# B&R Automation Studio project Soiled_PLC (part 10)

#### Param_1_5kwStar.dat
```
(********************************************************************
 * COPYRIGHT --
 ********************************************************************
 * Data object: Param_1_5kwStar
 * File: Param_1_5kwStar.dat
 * Author:  D.Jefferys
 * Created: October 2, 2009
 ********************************************************************
 * Data object file: Param_1_5kwStar.dat
 ********************************************************************)

;Version 2.00 18/10/2010 D.J. Added 14-26 Trip Delay - Disabled, Changed 14-10 from 3 (Coasting) to 5 (Kenetic Backup + Trip)
;Version 3.00 03/11/2010 D.J. Added CAN Switch Settings
;Version 4.00 02/11/2011 D.J. Added Parameter 40 - Hand on Key on LCP now Disabled

;CAN Module Switch Settings
;--------------------------

;Baudrate
;8 on  7 on  Par 10-01
;8 on  7 off 500kbps
;8 off 7 on  250kbps
;8 off 7 off 125kbps

;Node Number Binary
;1 = 1s
;2 = 2s
;3 = 4s
;4 = 8s
;5 = 16s
;6 = 32s

;
;	!!! DO NOT CHANGE THE SEQUENCE OF THE PARAMETERS
;
; FU parameter to the Ubertragung (only parameter, which deviates from the default values)
;
; 1.5 kW Star
;
; Index, Subindex, Datatype (Bytes), Setting (DINT) ; Comments
0002,00,01,00000001	; [000] 00-02, Motor Speed 0 - RPM, 1 - Hz
0001,00,01,00000000	; [001] 00-01, Language 0 - English, 1 - German
0011,00,01,00000001	; [002] 00-11, Edit Setup 1
0190,00,01,00000000	; [003] 01-90, Motor Thermal Protection, 2 - Thermistor
0040,00,01,00000000 ; [---] 00-40, Hand On Key on LCP 0 - Disabled No Function
0381,00,04,00000050 ; [000] 03-81, QuickStop ramp time 100 - 1s
0458,00,01,00000001	; [004] 04-58, Missing motor phase function, 1 - Trip 100ms
0854,00,01,00000001	; [005] 08-54, Reversing select 1 - Bus only 3 - Bus and Terminal
0211,00,02,00000310	; [006] 02-11, Brake resistor 120 Ohm
0212,00,04,00001200	; [007] 02-12, Brake power limit 1200 Watt
0213,00,01,00000002	; [008] 02-13, Brake check 2 - Alarm
1426,00,01,00000000 ; [---] 14-26, Trip delay at inverter fault 0 = Disabled
0803,00,04,00000002 ; [000] 08-03, Control Word Timeout Time 10 = 1Sec
0804,00,01,00000002	; [009] 08-04, Control Word Timeout Function 2 - Stop with auto restart
0801,00,01,00000002	; [010] 08-01, Control Site, 2 - Controlword only
0223,00,01,00000005	; [011] 02-23, Active brake delay 0,3 s
1761,00,01,00000002	; [012] 17-61, Encoder Signal Monitoring (Encoder faulty), 2 - Trip Changed for testing.
1710,00,01,00000001	; [013] 17-10, Encoder Signal Type 1 - TTL
1711,00,02,00001024	; [014] 17-11, Encoder Resolution 1024 Pulse
0430,00,01,00000001 ; [015] 04-30, Motor Feedback Loss Function, 1 - Warning, 2* - Trip
0431,00,02,00000300 ; [016] 04-31, Motor Feedback Speed Error RPM, 0-600, 300*
0226,00,02,00005000	; [015] 02-26, Torque Ref, 50,00%
0228,00,02,00000200	; [016] 02-28, Gain Boost Factor, 2,00% 0-4% ***************************
0519,00,01,00000003	; [017] 05-19, Terminal 37 Safe Stop, 3 - Safe Stop Warning
0120,00,04,00000150	; [018] 01-20, Motor Power 1.5kW
0101,00,01,00000003	; [019] 01-01, Motor Control Principle, 3 - Flux with motor feedback
0122,00,02,00000400	; [020] 01-22, Motor voltage 400 V
0123,00,02,00000050	; [021] 01-23, Motor frequency 50 Hz
0162,00,02,00000100	; [022] 01-62, Slip compenstation 100%
0410,00,01,00000002	; [023] 04-10, Motor speed direction, 2 - both directions
0540,00,01,00000032	; [024] 05-40, [0] Relay 1 Function, 32 - Mech brake ctrl
0540,01,01,00000032	; [025] 05-40, [1] Relay 2 Function, 32 - Mech brake ctrl
0802,00,01,00000003 ; [---] 08-02, Control Site 3 - Option A CAN Bus
0102,00,01,00000002	; [026] 01-02, Flux Motor Feeback Source 2 - MCB102
0125,00,02,00001400	; [027] 01-25, Motor nominal speed 1440 rpm
0702,00,02,00000070	; [028] 07-02, Speed PID proportionl gain 0,070
0700,00,01,00000002	; [029] 07-00, Speed PID Feedback Source 2 - MCB102
0172,00,01,00000006	; [030] 01-72, Start function, 6 - Hoist Mech. Brake Rel
0210,00,01,00000001	; [031] 02-10, Brake Function, 1 - Resistor brake
1410,00,01,00000005	; [032] 14-10, Mains failure, 3 - Coasting 5 - Kenetic backup , trip
0193,00,01,00000002	; [040] 01-93, Thermistor source, 2 Analogue input 54 Source terminal 50 for 10V //6 - Digital Input 33
0100,00,01,00000001	; [034] 01-00, Configuration mode, 1 - Closed loop with encoder
0139,00,01,00000004	; [035] 01-39, Motor poles, 4
0511,00,01,00000000	; [036] 05-11, Terminal 19, 0 - No Operation
0512,00,01,00000000	; [037] 05-12, Terminal 27, 0 - No Operation
0513,00,01,00000000	; [038] 05-13, Terminal 29, 0 - No Operation
0510,00,01,00000000	; [039] 05-10, Terminal 18, 0 - No Operation
0175,00,02,00000015	; [040] 01-75, Start Speed, 1,5 Hz
0222,00,02,00000005	; [041] 02-22, Activate Brake Speed ?en bei 0,5 Hz
0124,00,04,00000360	; [042] 01-24, Motor current 5,2 A
0341,00,04,00000100	; [043] 03-41, Ramp 1 ramp up time (1 Sec to 50 Hz)
0342,00,04,00000100	; [044] 03-42, Ramp 1 ramp down time (1 Sec to  0 Hz)
0414,00,02,00001000	; [045] 04-14, Motor Speed High Limit 100,0 Hz
0220,00,04,00000180	; [046] 02-20, Release brake current 1,8 A - About Half of motor A?
;0130,00,04,00029763	; [047] 01-30, Stator resistance (Rs) 2,9763 Ohm
;0131,00,04,00022212	; [048] 01-31, Rotor resistance (Rr) 2,2212 Ohm
;0134,00,04,00031036	; [049] 01-34, Rotor leakage reactance (X2) 3,1036 Ohm
;0136,00,04,01803904	; [050] 01-36, Iron loss resistance (Rfe) 1803,904 Ohm
;0135,00,04,00653996	; [051] 01-35, Main reactance (Xh) 65,3996 Ohm
0416,00,02,00002500	; [052] 04-16, Torque limit motor mode, 160,0 - % NOW 250%
0417,00,02,00001600	; [053] 04-17, Torque limit generator mode, 160,0 %
;0133,00,04,00031036	; [054] 01-33, Stator leakage reactance (X1), 3,1036 Ohm
0303,00,04,00100000	; [055] 03-03, Maximum Reference, 100,000
0418,00,04,00001720	; [056] 04-18, Current Limit 172,0 % - NOW 250%
```

### Data object Logical/Robo_Drive_Control/Paramaters_AnaloguePTC/Param_0_25kwStar1 (Simple, version 4.00.0) - Parameters 0.25kW Star Analogue PTC

#### Param_0_25kwStar.dat
```
(********************************************************************
 * COPYRIGHT --
 ********************************************************************
 * Data object: Param_2kwStar
 * File: Param_2kwStar.dat
 * Author:  D.Jefferys
 * Created: February 12, 2009
 ********************************************************************
 * Data object file: Param_2kwStar.dat
 ********************************************************************)

;Version 2.00 18/10/2010 D.J. Added 14-26 Trip Delay - Disabled, Changed 14-10 from 3 (Coasting) to 5 (Kenetic Backup + Trip)
;Version 3.00 03/11/2010 D.J. Added CAN Switch Settings
;Version 4.00 02/11/2011 D.J. Added Parameter 40 - Hand on Key on LCP now Disabled

;CAN Module Switch Settings
;--------------------------

;Baudrate
;8 on  7 on  Par 10-01
;8 on  7 off 500kbps
;8 off 7 on  250kbps
;8 off 7 off 125kbps

;Node Number Binary
;1 = 1s
;2 = 2s
;3 = 4s
;4 = 8s
;5 = 16s
;6 = 32s

;
;	!!! DO NOT CHANGE THE SEQUENCE OF THE PARAMETERS
;
; FU parameter to the Ubertragung (only parameter, which deviates from the default values)
;
; 0.25 kW Star
;
; Index, Subindex, Datatype (Bytes), Setting (DINT) ; Comments
0002,00,01,00000001	; [000] 00-02, Motor Speed 0 - RPM, 1 - Hz
0001,00,01,00000000	; [001] 00-01, Language 0 - English, 1 - German
0011,00,01,00000001	; [002] 00-11, Edit Setup 1
;0190,00,01,00000000	; [003] 01-90, Motor Thermal Protection, 0 - No protection
0040,00,01,00000000 ; [---] 00-40, Hand On Key on LCP 0 - Disabled No Function
0381,00,04,00000050 ; [000] 03-81, QuickStop ramp time 100 - 1s
;0458,00,01,00000001	; [004] 04-58, Missing motor phase function, 1 - Trip 100ms
0854,00,01,00000001	; [005] 08-54, Reversing select 1 - Bus only 3 - Bus and Terminal
0211,00,02,00000620	; [006] 02-11, Brake resistor 620 Ohm
0212,00,04,00000065	; [007] 02-12, Brake power limit 65 Watt
0213,00,01,00000002	; [008] 02-13, Brake check 2 - Alarm
1426,00,01,00000000 ; [---] 14-26, Trip delay at inverter fault 0 = Disabled
0803,00,04,00000002 ; [000] 08-03, Control Word Timeout Time 10 = 1Sec
0804,00,01,00000002	; [009] 08-04, Control Word Timeout Function 2 - Stop with auto restart
0801,00,01,00000002	; [010] 08-01, Control Site, 2 - Controlword only
0223,00,01,00000005	; [011] 02-23, Active brake delay 0,3 s
1761,00,01,00000002	; [012] 17-61, Encoder Signal Monitoring (Encoder faulty), 2 - Trip
1710,00,01,00000001	; [013] 17-10, Encoder Signal Type 1 - TTL
1711,00,02,00001024	; [014] 17-11, Encoder Resolution 1024 Pulse
0430,00,01,00000001 ; [015] 04-30, Motor Feedback Loss Function, 1 - Warning, 2* - Trip
0431,00,02,00000600 ; [016] 04-31, Motor Feedback Speed Error RPM, 0-600, 300*
0226,00,02,00005000	; [017] 02-26, Torque Ref, 50,00%
0228,00,02,00000200	; [018] 02-28, Gain Boost Factor, 2,00% 0-4% ***************************
0519,00,01,00000003	; [019] 05-19, Terminal 37 Safe Stop, 3 - Safe Stop Warning
0120,00,04,00000025	; [020] 01-20, Motor Power 0.25kW
0101,00,01,00000003	; [021] 01-01, Motor Control Principle, 3 - Flux with motor feedback
0122,00,02,00000400	; [022] 01-22, Motor voltage 400 V
0123,00,02,00000050	; [023] 01-23, Motor frequency 50 Hz
0162,00,02,00000100	; [024] 01-62, Slip compenstation 100%
0410,00,01,00000002	; [025] 04-10, Motor speed direction, 2 - both directions
0540,00,01,00000032	; [026] 05-40, [0] Relay 1 Function, 32 - Mech brake ctrl
0540,01,01,00000032	; [027] 05-40, [1] Relay 2 Function, 32 - Mech brake ctrl
0802,00,01,00000003 ; [---] 08-02, Control Site 3 - Option A CAN Bus
0102,00,01,00000002	; [028] 01-02, Flux Motor Feeback Source 2 - MCB102
0125,00,02,00001350	; [029] 01-25, Motor nominal speed 1350 rpm
0702,00,02,00000040	; [030] 07-02, Speed PID proportionl gain 0,040
0700,00,01,00000002	; [031] 07-00, Speed PID Feedback Source 2 - MCB102
0172,00,01,00000006	; [032] 01-72, Start function, 6 - Hoist Mech. Brake Rel
0210,00,01,00000001	; [033] 02-10, Brake Function, 1 - Resistor brake
1410,00,01,00000005	; [034] 14-10, Mains failure, 3 - Coasting 5 - Kenetic backup , trip
0193,00,01,00000002	; [040] 01-93, Thermistor source, 2 Analogue input 54 Source terminal 50 for 10V //6 - Digital Input 33
0100,00,01,00000001	; [036] 01-00, Configuration mode, 1 - Closed loop with encoder
0139,00,01,00000004	; [037] 01-39, Motor poles, 4
0511,00,01,00000000	; [038] 05-11, Terminal 19, 0 - No Operation
0512,00,01,00000000	; [039] 05-12, Terminal 27, 0 - No Operation
0513,00,01,00000000	; [040] 05-13, Terminal 29, 0 - No Operation
0510,00,01,00000000	; [041] 05-10, Terminal 18, 0 - No Operation
0175,00,02,00000015	; [042] 01-75, Start Speed, 1,5 Hz
0222,00,02,00000005	; [043] 02-22, Activate Brake Speed ?en bei 0,5 Hz
0124,00,04,00000089	; [044] 01-24, Motor current 0,89 A
0341,00,04,00000100	; [045] 03-41, Ramp 1 ramp up time (1 Sec to 50 Hz)
0342,00,04,00000100	; [046] 03-42, Ramp 1 ramp down time (1 Sec to  0 Hz)
0414,00,02,00001000	; [047] 04-14, Motor Speed High Limit 100,0 Hz
;0220,00,04,00000260	; [048] 02-20, Release brake current 2,6 A
;0130,00,04,00029763	; [049] 01-30, Stator resistance (Rs) 2,9763 Ohm
;0131,00,04,00022212	; [050] 01-31, Rotor resistance (Rr) 2,2212 Ohm
;0132,00,04,00031036	; [051] 01-34, Rotor leakage reactance (X2) 3,1036 Ohm
;0136,00,04,01803904	; [052] 01-36, Iron loss resistance (Rfe) 1803,904 Ohm
;0135,00,04,00653996	; [053] 01-35, Main reactance (Xh) 65,3996 Ohm
0416,00,02,00001600	; [054] 04-16, Torque limit motor mode, 160,0 %
0417,00,02,00001600	; [055] 04-17, Torque limit generator mode, 160,0 %
;0133,00,04,00031036	; [056] 01-33, Stator leakage reactance (X1), 3,1036 Ohm
0303,00,04,00050000	; [057] 03-03, Maximum Reference, 100,000 50,000 Rotate for now!
0418,00,04,00001720	; [058] 04-18, Current Limit 172,0 %
```

- Data object Logical/Robo_Drive_Control/Param_3kw (Simple, version 4.00.0) - Parameters 3kW Star from Expo (no source held here)

- Data object Logical/Robo_Drive_Control/Param_1_5kwStar (Simple, version 4.00.1) - Parameters 1.5kW Star (no source held here)

- Program Logical/Robo_Drive_Control/zzRoboPosnNames (IEC) - Robo Position Names - Transfer TrackView (no source held here)

- Program Logical/Robo_Drive_Control/zzRoboPosnNamesTest (IEC) - Robo Position Names Test (no source held here)

- Program Logical/Robo_Drive_Control/Lift_PosMonitor (IEC) - *1ms Task to monitor and auto reference VC Works with liftv7 (no source held here)

### Program Logical/Robo_Drive_Control/Lift_v8_1 (IEC, version 8.00.2)

#### Lift.ab - Cyclic code
```automation-basic
;--------------------------------------
;Lift Drive Control - Original 2 Column
;--------------------------------------

;Version 1.00 23/02/2009 D.J. First Issue
;Version 2.00 03/11/2010 D.J. Changed RB to RB (Robo)
;Version 3.00 04/12/2010 D.J. New distance calculation by using encoder pulses for 1 meter
;Version 4.00 04/03/2011 D.J. Set RunHz to 0 when not on step 30
;Version 5.00 08/01/2013 T.R Add module OK to monitor Counter Card and force step 0 after error/powerup..Increased Param Count for Brake contact monitoring. Force init values when 0.
;Version 5.01 12/03/2013 T.R Change function of module OK monitoring to always restart seq after fail due to power cycles on remote panels.
;Version 6.01 			T.R Add Auto Reference function
;Version 6.02 27/11/2015 TR. Add Correct comments,
;Version V8 -- TR Send QS command when enable is off due to DANFOSS issues.

PROGRAM _INIT

 	;Set array index with each init call
	idx  = 0

	TaskNameID = ST_name(0,ADR(TaskName),0)

	IF (TaskNameID = 0) THEN
		TaskNameLen = strlen(ADR(TaskName))
		idx 		= UINT(atoi(ADR(TaskName) + (TaskNameLen - 1)))
	ENDIF

	RunTask = (idx > 0) and (idx <= (SIZEOF(RB)/SIZEOF(RB[0])))

	IF RunTask THEN

		;Calculate in future for different arrangements
		;----------------------------------------------

		;New calculation based on measuring the pulsed for 1000 mm of Travel
		;-------------------------------------------------------------------

		;Pulses per meter = 122864.6
		;My Ratio (Gearbox and Cog combined) = 4096 / 122.8646 = 33.3375
		;mm/minute 				= Motor Nominal Speed 1500 * My Ratio = 50006.25
		;mm/sec @ 50 Hz 		= 833.4375
		;mm/Hz 	833.4375 / 50 	= 16.6687

		RB[idx].Lift.PulsePer10th_mm = REAL(12.2865)
		RB[idx].Lift.mmPerHz = 16.6687
		;Force Init value if 0
		IF RB_Posn[idx].Lift.RefOffset = 0 THEN
			RB_Posn[idx].Lift.RefOffset = 20000 ; 2metres
		ENDIF
		IF RB_Posn[idx].Lift.MaxSpeed = 0 THEN
			RB_Posn[idx].Lift.MaxSpeed = 200
		ENDIF
	ENDIF

	STEP 					= 0
	RB[idx].Lift.SeqStep	= 0
	RetryCount				= 0

END_PROGRAM
PROGRAM _CYCLIC

	;----
	;Lift
	;----

	myStatus = FC302_SEQ_OK

	;CAN node, Parameter Table Name and IF address
	node 	= RB[idx].Lift.SeqIn.Node
	strcpy(ADR(sTableName),ADR(RB[idx].Lift.SeqIn.sParTblName))
	strcpy(ADR(sDevice),ADR(RB[idx].Lift.SeqIn.sDevice))

	RB[idx].Lift.SeqIn.I_RefPosn  = X[30 + (idx * 2)].X04

	;Read drive status
	FC302_ReadSTW_0.StatusWord = RB[idx].Lift.CAN.StatusWord
	FC302_ReadSTW_0 FUB FC302_ReadSTW()
	RB[idx].Lift.STW = FC302_ReadSTW_0.STW

	;Clear control word - drive stopped
	RB[idx].Lift.CTW.ExtRefSelectionLSB 	= FALSE
	RB[idx].Lift.CTW.ExtRefSelectionMSB 	= FALSE
	RB[idx].Lift.CTW.DC_Brake				= FALSE
	RB[idx].Lift.CTW.Coasting				= FALSE
	RB[idx].Lift.CTW.QuickStop				= FALSE
	RB[idx].Lift.CTW.HoldOutputFreq			= FALSE
	RB[idx].Lift.CTW.RampStopStart			= FALSE
	RB[idx].Lift.CTW.ResetTrip				= ResetTrip
	RB[idx].Lift.CTW.Jog					= FALSE
	RB[idx].Lift.CTW.RampSelection			= FALSE
	RB[idx].Lift.CTW.DataValid				= TRUE
	RB[idx].Lift.CTW.Relay01Active			= FALSE
	RB[idx].Lift.CTW.Relay02Active			= FALSE
	RB[idx].Lift.CTW.ParaSetUpLSB			= FALSE
	RB[idx].Lift.CTW.ParaSetUpMSB			= FALSE
	RB[idx].Lift.CTW.Reverse				= FALSE

	RB[idx].Lift.RunForwards				= FALSE
	RB[idx].Lift.RunReverse					= FALSE
	RB[idx].Lift.CAN.TargetVelocity			= 0
	RB[idx].Lift.RunFreq 					= 0
	RB[idx].Lift.SeqOut.RefComplete 		= FALSE
	RB[idx].Lift.SeqOut.PosnOk				= FALSE
	RB[idx].Lift.SeqOut.DriveDisabled		= FALSE
	Referencing								= FALSE
	DisableDrive 							= (RB[idx].Lift.SeqIn.DisableDrive OR RB[idx].Lift.SeqIn.EStop OR NOT RB[idx].Lift.STW.DriveReady OR NOT RB[idx].Lift.ModuleOK)
	LimitsOk								= (RB[idx].Lift.SeqIn.I_ForwardLimitOk AND RB[idx].Lift.SeqIn.I_ReverseLimitOk)
	ManualControl							= (RB_Posn[idx].Lift.OperationMode = 1)

	;Init var ensure not lost if no Init
	RB[idx].Lift.PulsePer10th_mm 			= REAL(12.2865)
	RB[idx].Lift.mmPerHz 					= 16.6687

	;Current Position
	RB[idx].Lift.PosnActRaw = (RB[idx].Lift.Encoder + $7FFFFFFF)
	RB[idx].Lift.PosnAct	= DINT(RB[idx].Lift.PosnActRaw / RB[idx].Lift.PulsePer10th_mm)
	RB[idx].Lift.PosnNow	= ((RB_Retain[idx].Lift.PosnRef - RB[idx].Lift.PosnAct) + RB_Posn[idx].Lift.RefOffset)
	RB[idx].Lift.DistRemain = ABS(RB[idx].Lift.SeqIn.PosnReq - RB[idx].Lift.PosnNow)

	;TrackView Display
	RB_Posn[idx].Lift.PositionNow 	= RB[idx].Lift.PosnNow
	RB_Posn[idx].Lift.CycleCount 	= RB_Perm[idx].Lift.CycleCount

	;Step Shifting
	STEP = RB[idx].Lift.SeqStep
	RB_Posn[idx].Lift.SeqStep = DINT(STEP)

	;Enable Parameter writing slower speed - Every 60ms
	ScanClock 		= clock_ms()
	ScanNow 		= (ScanClock - ScanLastClock)
	ScanLastClock 	= ScanClock
	ScanCount 		= (ScanCount + UINT(ScanNow))
	IF (ScanCount >= 60) THEN
		ScanCount = 0
	ENDIF
	ParameterEnable = (ScanCount = 0)

	;If ModuleOK Fails force reference.// Change to restart to CAN Sequence to ensure full control and correct params
;	F_TRIG(RB[idx].Lift.ModuleOK,CountCardFailedPLS)
;	IF CountCardFailedPLS AND (RetryCount < 5) THEN
;		RetryCount = RetryCount + 1  ;If required limit number of retries on the reference TEST IF REQUIRED> HOW TO HANDLE ERROR??
;		RB[idx].Lift.SeqIn.DoRef = TRUE
;	ENDIF
	IF NOT RB[idx].Lift.ModuleOK THEN	; Code to disable drive if count card failed/poweroff.
		RB[idx].Lift.SeqStep = 0
	ENDIF

	;Step 0 ;Disabled
	IF (STEP = 0) THEN
		IF (RunTask AND RB[idx].Lift.ModuleOK) THEN
			RB[idx].Lift.SeqStep = 1
		ELSE
			;Do Nothing
		ENDIF
	ENDIF

	;Set CAN node to pre-operational
	TON_10ms_Restart.IN = (STEP = 1)
	TON_10ms_Restart.PT = 1000
	TON_10ms_Restart FUB TON_10ms()
	IF (STEP = 1) THEN

		IF (StartNode = node) THEN
			StartNode = 0
		ENDIF

		myStatus = FC302_SEQ_SetCANPreOperational

		IF (RB[idx].Lift.CAN.ModuleOk OR (RB[idx].Lift.CAN.NodeStatus = 3)) THEN

			CANopenNMT_0.enable 	= TRUE
			CANopenNMT_0.pDevice 	= ADR(sDevice)
			CANopenNMT_0.node 		= node
			CANopenNMT_0.state 		= coENTER_PRE_OPERATIONAL
			CANopenNMT_0 FUB CANopenNMT()

			IF (CANopenNMT_0.status = 0) OR (CANopenNMT_0.status < 65535) THEN
				RB[idx].Lift.SeqStep = 10
			ENDIF

		ELSE IF TON_10ms_Restart.Q THEN
			RB[idx].Lift.SeqStep = 2 ;Reset node here if not true
		ENDIF

	ENDIF

	;Restart node
	IF (STEP = 2) THEN

		myStatus = FC302_SEQ_RestartCANnode

		CANopenNMT_0.enable 	= TRUE
		CANopenNMT_0.pDevice 	= ADR(sDevice)
		CANopenNMT_0.node 		= node
		CANopenNMT_0.state 		= coRESET_NODE
		CANopenNMT_0 FUB CANopenNMT()

		IF (CANopenNMT_0.status = 0) OR (CANopenNMT_0.status < 65535) THEN
			RB[idx].Lift.SeqStep = 1
		ENDIF

	ENDIF

	;Read from parameter table
	IF (STEP = 10) THEN

		myStatus = FC302_SEQ_ReadParameterTable

		TableTooLarge = FALSE

		FC302_ReadParamTbl_0.Enable 		= TRUE
		FC302_ReadParamTbl_0.adrTableName 	= ADR(sTableName)
		FC302_ReadParamTbl_0.adrDestTable 	= ADR(RB[idx].Lift.ParaList)
		FC302_ReadParamTbl_0.ParamLimit 	= (SIZEOF(RB[idx].Lift.ParaList) / 8)
		FC302_ReadParamTbl_0 FUB FC302_ReadParamTbl()

		IF FC302_ReadParamTbl_0.Status = 0 THEN
			WriteListLength = FC302_ReadParamTbl_0.ParamCount	;Total parameters to write to the drive
			WriteIndex 		= 0 								;First index to write 0 not used
			RB[idx].Lift.SeqStep = 11
		ELSE IF FC302_ReadParamTbl_0.Status = 1 THEN
			TableTooLarge = TRUE
		ELSE
			;Error
		ENDIF

	ENDIF

	;Write parameter list to drive
	IF (STEP = 11) THEN

		myStatus = FC302_SEQ_WriteParameters

		IF ParameterEnable THEN

			FC302_WriteParam_0.enable 	= TRUE
			FC302_WriteParam_0.pDevice 	= ADR(sDevice)
			FC302_WriteParam_0.node 	= node
			FC302_WriteParam_0.index 	= RB[idx].Lift.ParaList[WriteIndex].index
			FC302_WriteParam_0.subindex = RB[idx].Lift.ParaList[WriteIndex].subindex
			FC302_WriteParam_0.data 	= RB[idx].Lift.ParaList[WriteIndex].data
			FC302_WriteParam_0.bytelen 	= RB[idx].Lift.ParaList[WriteIndex].datalen
			FC302_WriteParam_0 FUB FC302_WriteParam()

			IF (FC302_WriteParam_0.status = 0) THEN
				RB[idx].Lift.SeqStep = 12
			ENDIF

		ENDIF

	ENDIF

	;Read Parameter from drive
	IF (STEP = 12) THEN

		myStatus = FC302_SEQ_WriteParameters

		IF ParameterEnable THEN

			FC302_ReadParam_0.enable 	= TRUE
			FC302_ReadParam_0.pDevice 	= ADR(sDevice)
			FC302_ReadParam_0.node 		= node
			FC302_ReadParam_0.index 	= RB[idx].Lift.ParaList[WriteIndex].index
			FC302_ReadParam_0.subindex 	= RB[idx].Lift.ParaList[WriteIndex].subindex
			FC302_ReadParam_0 FUB FC302_ReadParam()

			IF (FC302_ReadParam_0.status = 0) THEN
				myRead 	= UDINT(FC302_ReadParam_0.data)
				IF RB[idx].Lift.ParaList[WriteIndex].data = myRead THEN
					WriteIndex = WriteIndex + 1
					;Once = all parameters have been completed as 60 = 0-59
					IF (WriteIndex = WriteListLength) THEN
						RB[idx].Lift.SeqStep = 13
					ELSE
						RB[idx].Lift.SeqStep = 11 ;Write Next Parameter
					ENDIF
				ELSE
					RB[idx].Lift.ParamWrite.ErrorCount 	= RB[idx].Lift.ParamWrite.ErrorCount + 1
					RB[idx].Lift.ParamWrite.Index 		= RB[idx].Lift.ParaList[WriteIndex].index
					RB[idx].Lift.ParamWrite.SubIndex 	= RB[idx].Lift.ParaList[WriteIndex].subindex
					RB[idx].Lift.SeqStep = 11 ;Try Write Again
				ENDIF
			ENDIF

		ENDIF

	ENDIF

	;Store Parameters
	IF (STEP = 13) THEN

		myStatus = FC302_SEQ_WriteParameters

		IF ParameterEnable THEN

			FC302_WriteParam_0.enable 	= TRUE
			FC302_WriteParam_0.pDevice 	= ADR(sDevice)
			FC302_WriteParam_0.node 	= node
			FC302_WriteParam_0.index 	= 1031
			FC302_WriteParam_0.subindex = 0
			FC302_WriteParam_0.data 	= 1
			FC302_WriteParam_0.bytelen 	= 1
			FC302_WriteParam_0 FUB FC302_WriteParam()

			IF (FC302_WriteParam_0.status = 0) THEN
				RB[idx].Lift.SeqStep = 14
			ENDIF

		ENDIF

	ENDIF

	;Check Parameters are stored
	IF (STEP = 14) THEN

		myStatus = FC302_SEQ_CheckParamStored

		IF ParameterEnable THEN

			FC302_ReadParam_0.enable 	= TRUE
			FC302_ReadParam_0.pDevice 	= ADR(sDevice)
			FC302_ReadParam_0.node 		= node
			FC302_ReadParam_0.index 	= 1031
			FC302_ReadParam_0.subindex 	= 0
			FC302_ReadParam_0 FUB FC302_ReadParam()

			IF (FC302_ReadParam_0.status = 0) THEN
				IF (FC302_ReadParam_0.data = 0) THEN
					RB[idx].Lift.SeqStep = 15
				ENDIF
			ENDIF

		ENDIF

	ENDIF

	;Start CAN node
	IF (STEP = 15) THEN

		IF (StartNode = 0) THEN
			StartNode = node
		ENDIF

		IF (ParameterEnable AND (StartNode = node)) THEN

			myStatus = FC302_SEQ_StartCANnode

			CANopenNMT_0.enable 	= TRUE
			CANopenNMT_0.pDevice 	= ADR(sDevice)
			CANopenNMT_0.node 		= node
			CANopenNMT_0.state 		= coSTART_REMOTE_NODE
			CANopenNMT_0 FUB CANopenNMT()

			IF (CANopenNMT_0.status = 0) THEN
				RB[idx].Lift.SeqStep = 20
			ENDIF
		ENDIF

	ENDIF

	;Wait for drive operational
	TON_10ms_Retry.IN = (STEP = 20)
	TON_10ms_Retry.PT = 100 ;2000
	TON_10ms_Retry FUB TON_10ms()
	IF (STEP = 20) THEN
		myStatus = FC302_SEQ_WaitDriveOperational
		IF RB[idx].Lift.CAN.ModuleOk THEN
			IF (StartNode = node) THEN
				StartNode = 0
			ENDIF
			RB[idx].Lift.SeqStep 	= 21
		ELSE IF TON_10ms_Retry.Q THEN
			IF (StartNode = node) THEN
				StartNode = 0
			ENDIF
			RB[idx].Lift.SeqStep 	= 15 ;0
		ENDIF
	ENDIF

	;-----------------
	;Find ref Position
	;-----------------

	EnableReference = NOT DisableDrive

	;Past Reference position timer
	TON_10ms_PastRef.IN = NOT RB[idx].Lift.SeqIn.I_RefPosn
	TON_10ms_PastRef.PT = 30
	TON_10ms_PastRef FUB TON_10ms()

	RefSpeed = 100 ;150 ;15Hz

	;Move carriage down until refence or bottom limit
	IF (STEP = 21) THEN
		myStatus = FC302_SEQ_Referencing
		Referencing					= TRUE
		RB[idx].Lift.RunForwards 	= FALSE
		RB[idx].Lift.RunReverse 	= EnableReference
		RB[idx].Lift.RunFreq		= RefSpeed
		IF RB[idx].Lift.SeqIn.I_RefPosn THEN
			RB[idx].Lift.SeqStep = 23
		ELSE IF NOT RB[idx].Lift.SeqIn.I_ReverseLimitOk THEN
			RB[idx].Lift.SeqStep = 22
		ELSE IF NOT RB[idx].Lift.SeqIn.I_ForwardLimitOk THEN
			myStatus = FC302_SEQ_MotorWiringFault
		ENDIF
	ENDIF

	;Bottom limit was found - try moving up
	IF (STEP = 22) THEN
		myStatus = FC302_SEQ_Referencing
		Referencing					= TRUE
		RB[idx].Lift.RunForwards 	= EnableReference
		RB[idx].Lift.RunReverse 	= FALSE
		RB[idx].Lift.RunFreq		= RefSpeed
		IF RB[idx].Lift.SeqIn.I_RefPosn THEN
			RB[idx].Lift.SeqStep = 23
		ELSE IF NOT RB[idx].Lift.SeqIn.I_ForwardLimitOk THEN
			myStatus = FC302_SEQ_RefNotFound
		ENDIF
	ENDIF

	;Move carriage down past reference
	IF (STEP = 23) THEN
		myStatus = FC302_SEQ_Referencing
		Referencing					= TRUE
		RB[idx].Lift.RunForwards 	= FALSE
		RB[idx].Lift.RunReverse 	= EnableReference
		RB[idx].Lift.RunFreq		= RefSpeed
		IF TON_10ms_PastRef.Q THEN
			RB[idx].Lift.SeqStep = 24
		ENDIF
	ENDIF

	;Move carriage back up to reference
	IF (STEP = 24) THEN
		myStatus = FC302_SEQ_Referencing
		Referencing					= TRUE
		RB[idx].Lift.RunForwards 	= EnableReference
		RB[idx].Lift.RunReverse 	= FALSE
		RB[idx].Lift.RunFreq		= RefSpeed
		IF RB[idx].Lift.SeqIn.I_RefPosn THEN
			RB[idx].Lift.SeqStep = 25
		ENDIF
	ENDIF

	;Move carriage up clear of reference
	IF (STEP = 25) THEN
		myStatus = FC302_SEQ_Referencing
		Referencing					= TRUE
		RB[idx].Lift.RunForwards 	= EnableReference
		RB[idx].Lift.RunReverse 	= FALSE
		RB[idx].Lift.RunFreq		= 100
		IF TON_10ms_PastRef.Q THEN
			RB[idx].Lift.SeqStep = 26
		ENDIF
	ENDIF

	;Move carriage down until refence - final posioning
	IF (STEP = 26) THEN
		myStatus = FC302_SEQ_Referencing
		Referencing					= TRUE
		RB[idx].Lift.RunForwards 	= FALSE
		RB[idx].Lift.RunReverse 	= EnableReference
		RB[idx].Lift.RunFreq		= 10  ;1Hz get exact location
		IF RB[idx].Lift.SeqIn.I_RefPosn THEN
			RB_Retain[idx].Lift.PosnRef = RB[idx].Lift.PosnAct
			RB[idx].Lift.SeqStep = 30
		ENDIF
	ENDIF

	;------------------
	;Auto tune Position
	;------------------

	EnableTune = NOT DisableDrive

	;Rail in correct position proximity - depending on which is required
	I_InPosition = FALSE
	IF (RB[idx].Lift.SeqIn.AutoTuneReceive = AlignReceive) THEN
		I_InPosition = RB[idx].Lift.SeqIn.I_RailOkReceive
	ELSE
		I_InPosition = RB[idx].Lift.SeqIn.I_RailOkRelease
	ENDIF

	;Check in rough position Release or Recieve Prox Made
	IF (STEP = 41) THEN
		myStatus = FC302_SEQ_AutoTune
		RB[idx].Lift.SeqOut.AutoTunePosn = RB[idx].Lift.SeqIn.AutoTunePosn ;Auto Tune Status back to sequence
		IF I_InPosition THEN
			RB[idx].Lift.SeqStep = 42
		ELSE
			;Do What?
		ENDIF
		IF (RB[idx].Lift.SeqIn.AutoTunePosn = 0) THEN
			RB[idx].Lift.SeqStep = 30 ;Cancel AutoTune
		ENDIF
	ENDIF

	;Move up until prox not made and store value
	IF (STEP = 42) THEN
		myStatus = FC302_SEQ_AutoTune
		RB[idx].Lift.RunForwards 	= EnableTune
		RB[idx].Lift.RunReverse 	= FALSE
		RB[idx].Lift.RunFreq		= 10
		IF NOT I_InPosition THEN
			AutoSavedTop			= RB[idx].Lift.PosnNow
			RB[idx].Lift.SeqStep 	= 43
		ENDIF
		IF (RB[idx].Lift.SeqIn.AutoTunePosn = 0) THEN
			RB[idx].Lift.SeqStep = 30 ;Cancel AutoTune
		ENDIF
	ENDIF

	;Move down until prox made
	IF (STEP = 43) THEN
		myStatus = FC302_SEQ_AutoTune
		RB[idx].Lift.RunForwards 	= FALSE
		RB[idx].Lift.RunReverse 	= EnableTune
		RB[idx].Lift.RunFreq		= 10
		IF I_InPosition THEN
			RB[idx].Lift.SeqStep 	= 44
		ENDIF
		IF (RB[idx].Lift.SeqIn.AutoTunePosn = 0) THEN
			RB[idx].Lift.SeqStep = 30 ;Cancel AutoTune
		ENDIF
	ENDIF

	;Move down until prox not made and calc position difference
	IF (STEP = 44) THEN
		myStatus = FC302_SEQ_AutoTune
		RB[idx].Lift.RunForwards 	= FALSE
		RB[idx].Lift.RunReverse 	= EnableTune
		RB[idx].Lift.RunFreq		= 10
		IF NOT I_InPosition THEN
			AutoSavedBottom			= RB[idx].Lift.PosnNow
			RB[idx].Lift.SeqStep 	= 45
		ENDIF
		IF (RB[idx].Lift.SeqIn.AutoTunePosn = 0) THEN
			RB[idx].Lift.SeqStep = 30 ;Cancel AutoTune
		ENDIF
	ENDIF

	;Store new position
	IF (STEP = 45) THEN

		myStatus = FC302_SEQ_AutoTune

		;Calculate position
		AutoPosnDiff = ((AutoSavedTop - AutoSavedBottom) / 2)
		AutoNewPosn  = (AutoSavedTop - AutoPosnDiff)

		RB_Posn[idx].Lift.Posn[RB[idx].Lift.SeqIn.AutoTunePosn] = AutoNewPosn

		RB[idx].Lift.SeqOut.AutoTunePosn = 0 ;Clear Auto Position
		RB[idx].Lift.SeqStep = 46

	ENDIF

	;Wait until RB sequence has cancelled auto position
	IF (STEP = 46) THEN
		IF (RB[idx].Lift.SeqIn.AutoTunePosn = 0) THEN
			RB[idx].Lift.SeqStep = 30
		ENDIF
	ENDIF

	;Read a parameter - not used at present
	IF ((STEP < 11) OR (STEP > 14)) AND (RB[idx].Lift.CAN.ModuleOk OR (RB[idx].Lift.CAN.NodeStatus = 3)) THEN

		IF ParameterEnable THEN

			D[85] = MonitorIdx

			MonitorSubIndex = 0
			IF (MonitorIdx = 1) THEN
				MonitorIndex 	= 1610 ;Motor Power
			ELSE IF (MonitorIdx = 2) THEN
				MonitorIndex 	= 1612 ;Motor Voltage
			ELSE IF (MonitorIdx = 3) THEN
				MonitorIndex 	= 1613 ;Motor Hz
			ELSE IF (MonitorIdx = 4) THEN
				MonitorIndex 	= 1614 ;Motor A
			ELSE IF (MonitorIdx = 5) THEN
				MonitorIndex 	= 1616 ;Motor Torque Nm
			ELSE IF (MonitorIdx = 6) THEN
				MonitorIndex 	= 1617 ;Motor RPM
			ELSE IF (MonitorIdx = 7) THEN
				MonitorIndex 	= 1634 ;Drive °C
			ELSE IF (MonitorIdx = 8) THEN
				MonitorIndex 	= 1502 ;Motor kWh
			ELSE IF (MonitorIdx = 9) THEN
				MonitorIndex 	= 1690 ;Alarm word
			ELSE IF (MonitorIdx = 10) THEN
				MonitorIndex 	= 1691 ;Alarm word 2
			ELSE IF (MonitorIdx = 11) THEN
				MonitorIndex 	= 1692 ;Warning word
			ELSE IF (MonitorIdx = 12) THEN
				MonitorIndex 	= 1693 ;Warning word 2
			ELSE
				MonitorIdx = 1
			ENDIF

			;Monitor caused CAN problems do not use!!
			;----------------------------------------
			;FC302_ReadParam_0.enable 	= TRUE
			;FC302_ReadParam_0.pDevice 	= ADR(sDevice)
			;FC302_ReadParam_0.node 		= node
			;FC302_ReadParam_0.index 	= MonitorIndex
			;FC302_ReadParam_0.subindex 	= MonitorSubIndex
			;FC302_ReadParam_0 FUB FC302_ReadParam()

			;IF (FC302_ReadParam_0.status = 0) THEN
			;	myRead 	= UINT(FC302_ReadParam_0.data)
			;ENDIF

			RB[idx].Lift.Motor.Value = INT(myRead)
			RB_Posn[idx].Lift.Monitor = INT(myRead)

		ENDIF

	ENDIF

	;Normal Operation
	IF (STEP = 30) THEN

		IF (mySlowWindow = 0) THEN
			mySlowWindow = 500 ;200 ;1000
		ENDIF
		IF (myDist = 0) THEN
			myDist = 250 ;200
		ENDIF

		RB[idx].Lift.SeqOut.RefComplete = TRUE

		;Power Save mode changed - re-calculate run speed
		IF PowerSave <> RB[idx].Lift.SeqIn.PowerSave THEN
			RB[idx].Lift.RunHz 	= 0
			PowerSave 			= RB[idx].Lift.SeqIn.PowerSave
		ENDIF

		;Calculate the required speed and stop distance with each run signal
		IF RB[idx].Lift.SeqIn.Run THEN
			IF (RB[idx].Lift.RunHz = 0) THEN
				;Required speed
				MotorNomHz 				= 50	;Motor nominal speed 50Hz
				RampTime 				= 10 	;1.0 sec - Read value in future?
				RampDist				= ((MotorNomHz * RB[idx].Lift.mmPerHz) * RampTime) ;Nominal Ramp Dist @ 50Hz
				DistRemain				= RB[idx].Lift.DistRemain
				RampFactor 				= (DistRemain / RampDist) ;eg 500mm Remain / 620mm (RampDist @ 50Hz) = 0.8
				RequiredHz				= UINT((MotorNomHz * RampFactor) * 10)
				MaxHz					= UINT((RB[idx].Lift.SeqIn.MaxSpeed / RB[idx].Lift.mmPerHz) * 10)
				;Restrict speed to value from sequence or 1000mm/sec (80.6 Hz)
				;IF (MaxHz > 806) THEN
				;	MaxHz = 806
				;ENDIF
				IF (MaxHz > 1209) THEN
					MaxHz = 1209
				ENDIF
				IF (RequiredHz > MaxHz) THEN
					RB[idx].Lift.RunHz 	= MaxHz
				ELSE
					RB[idx].Lift.RunHz 	= RequiredHz
				ENDIF
				;Stop Distance
				;RB[idx].Lift.StopDist 	= (((RB[idx].Lift.RunHz * RB[idx].Lift.SeqIn.RunSpeed) * RampTime) / 1000)
				StopFactor				= (REAL(RB[idx].Lift.RunHz) / (MotorNomHz * 10))
				RunSpeed				= (StopFactor * (RampDist / 10))
				RB[idx].Lift.StopDist	= UDINT((RunSpeed * StopFactor) / 0.2)
				SlowWindow 				= mySlowWindow ;1000 ;10tenths mm - try lower larger than CAN scan time
				StopDist				= RB[idx].Lift.StopDist + SlowWindow
			ENDIF

		ELSE
			RB[idx].Lift.RunHz = 0
		ENDIF

		;Position Required?
		IF (RB[idx].Lift.DistRemain > StopDist) THEN
			RB[idx].Lift.RunFreq 	= RB[idx].Lift.RunHz
		ELSE IF (RB[idx].Lift.DistRemain > myDist) THEN ;200) THEN 	;100 = 10mm
			RB[idx].Lift.RunFreq = 81 					;8.1Hz = 100mm/sec
		ELSE IF (RB[idx].Lift.DistRemain > 5) 	THEN 	;5 = 0.5mm
			RB[idx].Lift.RunFreq = 12					;1.2Hz, 0.8Hz = 10mm/sec
		ELSE
			RB[idx].Lift.RunFreq = 0
		ENDIF

		;Final Ramp Time
		IF (RB[idx].Lift.RunFreq = RB[idx].Lift.RunHz) THEN
			RB[idx].Lift.RampStart 	= 0
			RB[idx].Lift.RampTime 	= 0
		ELSE IF (RB[idx].Lift.RunFreq > 0) THEN
			IF (RB[idx].Lift.RampStart = 0) THEN
				RB[idx].Lift.RampStart = clock_ms()
			ENDIF
		ELSE IF (RB[idx].Lift.RunFreq = 0) THEN
			IF (RB[idx].Lift.RampTime = 0) THEN
				RB[idx].Lift.RampTime = (clock_ms() - TIME(RB[idx].Lift.RampStart))
			ENDIF
			;Store Max final ramp time
			IF (RB[idx].Lift.RampTime > RB[idx].Lift.RampMax) THEN
				RB[idx].Lift.RampMax = RB[idx].Lift.RampTime
			ENDIF
		ENDIF

		RB[idx].Lift.RunForwards 	= (RB[idx].Lift.SeqIn.Run AND (RB[idx].Lift.PosnNow < RB[idx].Lift.SeqIn.PosnReq))
		RB[idx].Lift.RunReverse 	= (RB[idx].Lift.SeqIn.Run AND (RB[idx].Lift.PosnNow > RB[idx].Lift.SeqIn.PosnReq))

		;Check Rail Alignment Switches
		IF RB[idx].Lift.SeqIn.Run THEN
			IF NOT AlignSwitchCheck THEN
				AlignSwitchCheck 	= TRUE
				ReleaseSwitchOk 	= FALSE
				ReceiveSwitchOk		= FALSE
			ENDIF
		ELSE
			AlignSwitchCheck = FALSE
		ENDIF

		;Switches have gone off during operation
		IF NOT RB[idx].Lift.SeqIn.I_RailOkRelease THEN
			ReleaseSwitchOk = TRUE
		ENDIF

		IF NOT RB[idx].Lift.SeqIn.I_RailOkReceive THEN
			ReceiveSwitchOk = TRUE
		ENDIF
		;------------------------------

		RailAligned = FALSE
		IF (RB[idx].Lift.SeqIn.RailAlign = AlignNone) THEN
			RailAligned	= TRUE
		ELSE IF (RB[idx].Lift.SeqIn.RailAlign = AlignReceive) AND RB[idx].Lift.SeqIn.I_RailOkReceive THEN
			RailAligned	= TRUE
		ELSE IF (RB[idx].Lift.SeqIn.RailAlign = AlignRelease) AND RB[idx].Lift.SeqIn.I_RailOkRelease THEN
			RailAligned	= TRUE
		ENDIF
		PosnValid					= (RB[idx].Lift.DistRemain <= 10) ;10=1mm
		AlignSwitchesOk				= (ReleaseSwitchOk AND ReceiveSwitchOk)
		RB[idx].Lift.SeqOut.PosnOk  = ((RB[idx].Lift.RunFreq = 0) AND PosnValid AND RailAligned AND AlignSwitchesOk)

		IF ((RB[idx].Lift.RunFreq = 0) AND PosnValid) THEN
			IF NOT RailAligned THEN
				myStatus = FC302_SEQ_RailNotAligned
			ELSE IF NOT ReleaseSwitchOk THEN
				myStatus = FC302_SEQ_ReleaseSwitchFault
			ELSE IF NOT ReceiveSwitchOk THEN
				myStatus = FC302_SEQ_ReceiveSwitchFault
			ENDIF
		ENDIF

		;Reference Check - CHeck position when moving down onto reference switch..

		;Travel limit reached go-to reference
		;IF NOT LimitsOk THEN
		;	RB[idx].Lift.SeqStep = 0
		;ENDIF

		;No reference position then go-to reference
		IF (RB_Retain[idx].Lift.PosnRef = 0) THEN
			RB[idx].Lift.SeqStep = 0
		ENDIF

		;Go to Manual Jog
		IF (RB[idx].Lift.SeqIn.JogForwards OR RB[idx].Lift.SeqIn.JogReverse) THEN
			JogHz				 = 100
			RB[idx].Lift.SeqStep = 32
		ENDIF

		;Auto fine tune required?
		IF (RB[idx].Lift.SeqIn.AutoTunePosn > 0) THEN
			RB[idx].Lift.SeqStep = 41
		ENDIF

		;Drive disable request or e-stop from sequence
		IF DisableDrive THEN
			RB[idx].Lift.SeqStep = 31
		ENDIF

	ELSE
		RB[idx].Lift.RunHz = 0
	ENDIF ;\Step 30

	;Drive Disabled - RB Sequence stops drive operation
	IF (STEP = 31) THEN
		RB[idx].Lift.SeqOut.RefComplete 	= TRUE
		RB[idx].Lift.SeqOut.DriveDisabled 	= DisableDrive
		IF NOT DisableDrive THEN
			RB[idx].Lift.SeqStep = 30
		ENDIF
	ELSE IF Referencing THEN
		RB[idx].Lift.SeqOut.DriveDisabled 	= DisableDrive
	ENDIF

	;RB Seq Do Reference Received
	IF (STEP <> 31) THEN
		IF RB[idx].Lift.SeqIn.DoRef THEN
			RB[idx].Lift.SeqIn.DoRef 	= FALSE
			IF (RB[idx].Lift.CAN.NodeStatus = 261) THEN
				RB[idx].Lift.SeqStep = 21
			ELSE
				RB[idx].Lift.SeqStep = 0
			ENDIF
		ENDIF
	ENDIF

	;Enable reset of drive when in error - trip lock and drive not ready etc..
	IF ((STEP = 31) AND NOT RB[idx].Lift.SeqIn.DisableDrive) THEN
		IF RB[idx].Lift.SeqIn.DoRef THEN
			RB[idx].Lift.SeqIn.DoRef 	= FALSE
			RB[idx].Lift.SeqStep 		= 0
		ENDIF
	ENDIF

	;Jog mode - 1 second slow before accelleration
	TmrJog.IN = (STEP = 32)
	TmrJog.PT = 100
	TmrJog FUB TON_10ms()
	IF (STEP = 32) THEN
		myStatus = FC302_SEQ_Jog
		Referencing					= TRUE
		RB[idx].Lift.RunForwards 	= RB[idx].Lift.SeqIn.JogForwards
		RB[idx].Lift.RunReverse 	= RB[idx].Lift.SeqIn.JogReverse
		RB[idx].Lift.RunFreq		= (JogHz / 10)
		IF (TmrJog.Q AND (JogHz < 1600)) THEN ;160 (1600 / 10) around 200mm/sec
			JogHz = JogHz + 1 ;Acc by 0.1 Hz / Scan 81 = 8.1Hz = 100mm/sec
		ENDIF
		IF (NOT RB[idx].Lift.SeqIn.JogForwards AND NOT RB[idx].Lift.SeqIn.JogReverse) THEN
			RB[idx].Lift.SeqStep = 30
		ENDIF
	ENDIF

	EnableForwards 	= (RB[idx].Lift.RunForwards AND RB[idx].Lift.SeqIn.I_ForwardLimitOk)
	EnableReverse	= (RB[idx].Lift.RunReverse  AND RB[idx].Lift.SeqIn.I_ReverseLimitOk)

	EnableDrive 	= (NOT DisableDrive AND (EnableForwards OR EnableReverse) AND (RB[idx].Lift.RunFreq > 0))

	QuickStop		= (RB[idx].Lift.SeqIn.EStop OR (NOT Referencing AND (NOT RB[idx].Lift.SeqIn.I_ForwardLimitOk OR NOT RB[idx].Lift.SeqIn.I_ReverseLimitOk)))
	;QuickStop		= RB[idx].Lift.SeqIn.EStop

	;Estop
	;Drive ready from status word and bus control

	;Give current position to RB sequence
	RB[idx].Lift.SeqOut.PosnNow = INT(RB[idx].Lift.PosnNow / 10)

	;Drive Control Word
	IF RB[idx].Lift.CAN.ModuleOk THEN
		IF EnableDrive AND NOT QuickStop THEN
			RB[idx].Lift.CTW.DC_Brake		= TRUE
			RB[idx].Lift.CTW.Coasting		= TRUE
			RB[idx].Lift.CTW.QuickStop		= (RB[idx].Lift.RunFreq > 0)
			RB[idx].Lift.CTW.HoldOutputFreq	= TRUE
			RB[idx].Lift.CTW.RampStopStart	= TRUE
			RB[idx].Lift.CTW.ResetTrip		= FALSE
			RB[idx].Lift.CTW.DataValid		= TRUE
			RB[idx].Lift.CTW.Reverse		= EnableForwards  	;Due to mechanical arrangement Reverse is Up/Forwards
			RB[idx].Lift.CAN.TargetVelocity	= UINT(($4000 / 1000) * RB[idx].Lift.RunFreq)
		ELSE
			RB[idx].Lift.CTW.DC_Brake		= FALSE//TRUE
			RB[idx].Lift.CTW.Coasting		= TRUE
			RB[idx].Lift.CTW.QuickStop		= FALSE// NOT QuickStop ;0 = QuickStop
			RB[idx].Lift.CTW.HoldOutputFreq	= FALSE//TRUE
			RB[idx].Lift.CTW.RampStopStart	= FALSE
			RB[idx].Lift.CTW.ResetTrip		= FALSE
			RB[idx].Lift.CTW.DataValid		= TRUE
			RB[idx].Lift.CTW.Reverse		= FALSE
			RB[idx].Lift.CAN.TargetVelocity	= $0000
		ENDIF
	ENDIF

	;Write control word to drive
	FC302_WriteCTW_0.CTW = RB[idx].Lift.CTW
	FC302_WriteCTW_0 FUB FC302_WriteCTW()
	RB[idx].Lift.CAN.ControlWord = FC302_WriteCTW_0.ControlWord

	;Scan time calculation
	IF NOT RB[idx].Lift.Scan.StartTrig AND NOT RB[idx].Lift.Scan.EndTrig THEN
		IF RB[idx].Lift.CTW.RampStopStart THEN
			RB[idx].Lift.Scan.Start 	= clock_ms()
			RB[idx].Lift.Scan.StartTrig = TRUE
		ENDIF
	ELSE IF RB[idx].Lift.Scan.StartTrig AND NOT RB[idx].Lift.Scan.EndTrig THEN
		IF RB[idx].Lift.STW.InOperation THEN
			RB[idx].Lift.Scan.End 		= clock_ms()
			RB[idx].Lift.Scan.EndTrig	= TRUE

			RB[idx].Lift.Scan.LastScan = UINT(RB[idx].Lift.Scan.End - RB[idx].Lift.Scan.Start)
			IF ((RB[idx].Lift.Scan.LastScan < RB[idx].Lift.Scan.MinScan) OR (RB[idx].Lift.Scan.MinScan = 0)) THEN
				RB[idx].Lift.Scan.MinScan = RB[idx].Lift.Scan.LastScan
			ENDIF
			IF (RB[idx].Lift.Scan.LastScan > RB[idx].Lift.Scan.MaxScan) THEN
				RB[idx].Lift.Scan.MaxScan = RB[idx].Lift.Scan.LastScan
			ENDIF
		ENDIF
	ELSE IF NOT RB[idx].Lift.CTW.RampStopStart AND NOT RB[idx].Lift.STW.InOperation THEN
		RB[idx].Lift.Scan.StartTrig = FALSE
		RB[idx].Lift.Scan.EndTrig 	= FALSE
	ENDIF

	;Status Word Warnings and Alarms
	IF RB[idx].Lift.STW.Trip THEN
		myStatus = FC302_STW_Trip
	ELSE IF RB[idx].Lift.STW.Error THEN
		myStatus = FC302_STW_Error
	ELSE IF RB[idx].Lift.STW.TripLock THEN
		myStatus = FC302_STW_TripLock
	ELSE IF RB[idx].Lift.STW.Warning THEN
		myStatus = FC302_STW_Warning
	ELSE IF RB[idx].Lift.STW.DriveOverTemp THEN
		myStatus = FC302_STW_DriveOverTemp
	ELSE IF RB[idx].Lift.STW.DriveVoltageFault THEN
		myStatus = FC302_STW_DriveVoltageFault
	ELSE IF RB[idx].Lift.STW.DriveTorqueLimit THEN
		myStatus = FC302_STW_DriveTorqueLimit
	ELSE IF RB[idx].Lift.STW.ThermalTimerLimit THEN
		myStatus = FC302_STW_ThermalTimeLimit
	ENDIF

	RB[idx].Lift.SeqOut.Status = myStatus

	;I/O Status to TrackView
	;-----------------------

	;Lift
	RB_Posn[idx].Lift.IOStatus  = 0 ;Clear
	IF RB[idx].Lift.SeqIn.I_RefPosn THEN
		RB_Posn[idx].Lift.IOStatus = BIT_SET(RB_Posn[idx].Lift.IOStatus, 0)
	ENDIF
	IF NOT RB[idx].Lift.SeqIn.I_ForwardLimitOk THEN
		RB_Posn[idx].Lift.IOStatus = BIT_SET(RB_Posn[idx].Lift.IOStatus, 1)
	ENDIF
	IF NOT RB[idx].Lift.SeqIn.I_ReverseLimitOk THEN
		RB_Posn[idx].Lift.IOStatus = BIT_SET(RB_Posn[idx].Lift.IOStatus, 2)
	ENDIF
	IF RB[idx].Lift.SeqIn.I_RailOkRelease THEN
		RB_Posn[idx].Lift.IOStatus = BIT_SET(RB_Posn[idx].Lift.IOStatus, 3)
	ENDIF
	IF RB[idx].Lift.SeqIn.I_RailOkReceive THEN
		RB_Posn[idx].Lift.IOStatus = BIT_SET(RB_Posn[idx].Lift.IOStatus, 4)
	ENDIF

END_PROGRAM
```

### Package Logical/KanLink_A19/Supertrack_Kanlink_Constants - *Kanlink constants

### KanLink_A19.typ - Global data types
```iecst
(********************************************************************
 * COPYRIGHT -- HP
 ********************************************************************
 * Package: KanLink_A7
 * File: KanLink_A7.typ
 * Author: treamsbottom
 * Created: January 28, 2013
 ********************************************************************
 * Data types of package KanLink_A7
 ********************************************************************)

TYPE
	IP_Type : 	STRUCT
		Area : UINT;
		Adr : UINT;
		CmdOpt : UINT;
		AdvMode : BOOL;
		AdrAdvMode : STRING[15];
	END_STRUCT;
	KanOVClient_typ : 	STRUCT
		IP : ARRAY[0..HLKANLINK_MAX_CLIENTCONNS]OF IP_Type;
		Enable : BOOL;
		MaxConns : UINT;
		InfoReq : ARRAY[0..HLKANLINK_MAX_CLIENTCONNS]OF BatchInfo_typ;
		InfoResp : ARRAY[0..HLKANLINK_MAX_CLIENTCONNS]OF InfoResp_typ;
		StatusReg : ARRAY[0..HLKANLINK_MAX_CLIENTCONNS]OF UINT;
		IndexOffset : UINT;
		CANOffset : UINT; (**Can offset for CAN live index passed to Tview*)
	END_STRUCT;
	KanOVServer_typ : 	STRUCT
		IP : ARRAY[0..HLKANLINK_MAX_SERVERCONNS]OF IP_Type;
		Enable : BOOL;
		MaxConns : UINT;
		InfoResp : ARRAY[0..HLKANLINK_MAX_SERVERCONNS]OF KLresp1002_Info_typ;
		IndexOffset : UINT;
	END_STRUCT;
	KanLinkCon_Typ : 	STRUCT
		Server : KANServer_typ;
		Client : KANClient_typ;
		OverviewServer : KanOVServer_typ;
		OverviewClient : KanOVClient_typ;
		ErrorString : STRING[80];
		GlobalSettings : KAN_Settings;
	END_STRUCT;
	KANClient_typ : 	STRUCT
		IP : ARRAY[0..HLKANLINK_MAX_CLIENTCONNS]OF IP_Type;
		Enable : BOOL;
		MaxConns : UINT;
		CANOffset : UINT;
	END_STRUCT;
	KANServer_typ : 	STRUCT
		IP : ARRAY[0..HLKANLINK_MAX_SERVERCONNS]OF IP_Type;
		Enable : BOOL;
		MaxConns : UINT;
		CANOffset : UINT;
		BagNum : ARRAY[0..HLKANLINK_MAX_SERVERCONNS]OF BagNums_typ;
	END_STRUCT;
	BagNums_typ : 	STRUCT
		BagNums : ARRAY[0..6]OF UINT;
	END_STRUCT;
	KANBatch_typ : 	STRUCT
		BatchData : ARRAY[0..6]OF BatchData_typ;
	END_STRUCT;
	BatchInfo_typ : 	STRUCT
		wCntPositions : UINT;
		wNoOfPosition : ARRAY[0..HLKANLINK_MAX_OVERVIEW_DATA]OF UINT;
		wRes : UINT;
	END_STRUCT;
	InfoResp_typ : 	STRUCT
		BagNum : ARRAY[0..HLKANLINK_MAX_OVERVIEW_DATA]OF UINT;
	END_STRUCT;
	KAN_Settings : 	STRUCT
		UseBatchCode : BOOL;
		TransferProgramCode : BOOL; (**This puts the cat code in custom area and transfers the prg code to the m/c*)
		BatchCodeTyp : USINT;
		TransferProgin_bCustom : BOOL;
	END_STRUCT;
END_TYPE
```

### KanLink_A19.var - Global variables
```iecst
(********************************************************************
 * COPYRIGHT -- HP
 ********************************************************************
 * Package: KanLink_A2
 * File: KanLink_A2.var
 * Author: treamsbottom
 * Created: September 07, 2012
 ********************************************************************
 * Variables of package KanLink_A2
 ********************************************************************)
VAR
	Kanlink : KanLinkCon_Typ; (**Configuration parameters*)
	PTResp : ARRAY[0..HLKANLINK_MAX_CLIENTCONNS] OF KL_BTxf_typ; (**Client comm var*)
	PT100 : ARRAY[0..HLKANLINK_MAX_SERVERCONNS] OF KL_BTxf_typ; (**Server comm var*)
	Batch : ARRAY[0..HLKANLINK_MAX_SERVERCONNS] OF KANBatch_typ;
	STOverReq : ARRAY[0..HLKANLINK_MAX_SERVERCONNS] OF KL_BI_typ; (*Overview Batch Info Server*)
	STOverResp : ARRAY[0..HLKANLINK_MAX_CLIENTCONNS] OF KL_BI_typ; (*Overview Batch Info Client*)
END_VAR
```

### Program Logical/KanLink_A19/zz_KanlinkConfig (IEC, version 1.20.0) - *Configuration of Kanlink

#### zz_KanlinkConfig.ab - Implementation code
```automation-basic
(********************************************************************
 * COPYRIGHT -- HP
 ********************************************************************
 * Program: zz_KanlinkConfig
 * File: zz_KanlinkConfig.ab
 * Author: treamsbottom
 * Created: September 07, 2012
 ********************************************************************
 * Implementation of program zz_KanlinkConfig
 ********************************************************************)
;Requirements
;From KGFramework
;	Libaries:
;		KgStdLib
;		KanLinkLib
;		mnParamLib
;	10ms Tasks:
;		hlKanLink
;	100ms Tasks:
;		svCPCache
;		mnEth
; When setting max connections for anything greater than 10
;the array decs will need changing. these are set by the constants HLKANLINK_MAX_CLIENTCONNS and HLKANLINK_MAX_SERVERCONNS in the frameworkshare
;Pkg_hlKanLink, KL_UserLib.Var
;----------------------------------------------------------------------------------------------------------------;
;-----21-1-2013..TR..Version A6 - First TestedVersion - Note Specials to run with Shuttle
;-----28-1-2013..TR..Version A7 - Remove Specials..Add option to send program and category number & Batch number.#
;-----03-03-2017..TR.Version A18 - Add "Advanced Connection Mode"
;-----07-06-2017 ..TR..Version A19 - Fix issues with sending empty bag date-- Remove reference to CAN[].Category -- Read all information from bag for consistency.
;-----------------------------------------------------------------------------------------------------------------

PROGRAM _CYCLIC
;HLKANLINK_MAX_SERVERCONNS	;Declaration of max Server conns for KG Framework
;HLKANLINK_MAX_CLIENTCONNS	;Declaration of max Client conns for KG Framework
IF NOT init THEN
;Parameter Setup
;Global setting - Apply to all Kanlink Comms(Server,Client,OverView)
	Kanlink.GlobalSettings.TransferProgramCode 	= FALSE ; This transfers/Read the cat code to/from the bCustom area. Prg to/from sCategory
	Kanlink.GlobalSettings.TransferProgin_bCustom = FALSE ;This transfers/Read the Program code to/from the bCustom area. Category to/from sCategory
	Kanlink.GlobalSettings.UseBatchCode 		= FALSE	; Pass batch/SQL id
	Kanlink.GlobalSettings.BatchCodeTyp			= BatchTyp_UDINT  ;0 = UDINT, 1 = 16 byte unique (UDINT By default, extra code required for 16 byte )

;---------------------------------------------------------Batch Transfer Server---------------------------------------------------------------
;Server (Used to send data)		--------------------------- Variable = PT100
	Kanlink.Server.Enable = TRUE ; used to enable Server Comms
	Kanlink.Server.MaxConns	= 1 ; Number of Server connections
	Kanlink.Server.CANOffset = 3 ; Start address of CAN variable
	;Address
	Kanlink.Server.IP[1].Area 	= 3 ;SDC1
	Kanlink.Server.IP[1].Adr 	= 13
	Kanlink.Server.IP[1].AdvMode = TRUE // Use Advance mode- Pass in whole IP address as a string.
	strcpy(ADR(Kanlink.Server.IP[1].AdrAdvMode),ADR("10.8.3.13"));

	Kanlink.Server.IP[1].CmdOpt = 0;
	Kanlink.Server.BagNum[1].BagNums[1] = 375 ; Bag number for data transfer
	Kanlink.Server.BagNum[1].BagNums[2] = 0 ; First buffer bag position ; Tunnel hasn't written code to recieve this yet..

		;---------------------------------------------------------Batch transfer Client---------------------------------------------------------------
	;Client used to recieve data --------------------------- Variable = PTResp
	Kanlink.Client.Enable = FALSE ; used to enable Client Comms
	Kanlink.Client.MaxConns	= 1 ; Number of Client connections
	Kanlink.Client.CANOffset = 21 ; Start address of CAN variable for the clients
	;Address
	Kanlink.Client.IP[1].Area 	= 1 ;Aero at sorting
	Kanlink.Client.IP[1].Adr 	= 91
	Kanlink.Client.IP[1].AdvMode = TRUE // Use Advance mode- Pass in whole IP address as a string.
	strcpy(ADR(Kanlink.Client.IP[1].AdrAdvMode),ADR("10.8.4.20"));

	Kanlink.Client.IP[1].CmdOpt = 0

;---------------------------------------------------------Overview Server---------------------------------------------------------------
	;------------------------------------------------Variable = STOverResp
	;Use Overview Server.. SendData Data to Overview PLC - Only IP necessary - Client will request bag numbers.
	Kanlink.OverviewServer.Enable = FALSE
	Kanlink.OverviewServer.MaxConns = 1

	Kanlink.OverviewServer.IP[1].Area = 4
	Kanlink.OverviewServer.IP[1].Adr = 21
	Kanlink.OverviewServer.IP[1].AdvMode = FALSE
	strcpy(ADR(Kanlink.OverviewServer.IP[1].AdrAdvMode),ADR("10.8.2.21"));

	Kanlink.OverviewServer.IP[1].CmdOpt = 0
;---------------------------------------------------------Overview Client---------------------------------------------------------------
;------------------------------------------------Variable = STOverReq
;Use Overview Client.. Recieve Data
	Kanlink.OverviewClient.Enable = FALSE
	Kanlink.OverviewClient.MaxConns = 5
	Kanlink.OverviewClient.CANOffset = 21
;-----------PLC 1 - AERO SYSTEM
	Kanlink.OverviewClient.StatusReg[1] = 951 ; D reg to map machine status for Tview.

	Kanlink.OverviewClient.IP[1].Area = 3
	Kanlink.OverviewClient.IP[1].Adr = 1	; To multiplex Edit KL_Overview
	Kanlink.OverviewClient.IP[1].AdvMode = FALSE
	strcpy(ADR(Kanlink.OverviewClient.IP[1].AdrAdvMode),ADR("10.8.3.1"));

	Kanlink.OverviewClient.IP[1].CmdOpt = 0
	//Batch data requested from Server
	Kanlink.OverviewClient.InfoReq[1].wCntPositions = 6  ;Number of positions requested max 6 per request. If more than 6 set to 0 to multiplex...
	Kanlink.OverviewClient.InfoReq[1].wNoOfPosition[0] = 1  ; Unqiue ID of data requested put all requests here if more than 6 the driver will multiplex the signals.
	Kanlink.OverviewClient.InfoReq[1].wNoOfPosition[1] = 2	; There must be no gaps in the request numbers.	If not multiplexing, ensure index[6] = 0
	Kanlink.OverviewClient.InfoReq[1].wNoOfPosition[2] = 3
	Kanlink.OverviewClient.InfoReq[1].wNoOfPosition[3] = 4
	Kanlink.OverviewClient.InfoReq[1].wNoOfPosition[4] = 5
	Kanlink.OverviewClient.InfoReq[1].wNoOfPosition[5] = 6

	//Bag number to map recieved data to.
	Kanlink.OverviewClient.InfoResp[1].BagNum[0] = 501
	Kanlink.OverviewClient.InfoResp[1].BagNum[1] = 502
	Kanlink.OverviewClient.InfoResp[1].BagNum[2] = 503
	Kanlink.OverviewClient.InfoResp[1].BagNum[3] = 504
	Kanlink.OverviewClient.InfoResp[1].BagNum[4] = 505
	Kanlink.OverviewClient.InfoResp[1].BagNum[5] = 506

;--------------------------------------------------------------END OF Configuration Code--------------------------------------------

;Check size of server and Client
	IF NOT Kanlink.Server.Enable THEN
		Kanlink.Server.MaxConns = 0
	ENDIF
	IF NOT Kanlink.Client.Enable THEN
		Kanlink.Client.MaxConns = 0
	ENDIF
	IF NOT Kanlink.OverviewServer.Enable THEN
		Kanlink.OverviewServer.MaxConns = 0
	ENDIF
	IF NOT Kanlink.OverviewClient.Enable THEN
		Kanlink.OverviewClient.MaxConns = 0
	ENDIF
	IF ((Kanlink.Server.MaxConns + Kanlink.OverviewServer.MaxConns) <= HLKANLINK_MAX_SERVERCONNS) THEN
		ServerDecOK = TRUE
	ELSE
		strcpy(ADR(Kanlink.ErrorString),"Declaration of HLKANLINK_MAX_SERVERCONNS not large enough")
		ServerDecOK = FALSE
	ENDIF
	IF ((Kanlink.Client.MaxConns + Kanlink.OverviewClient.MaxConns) <= HLKANLINK_MAX_CLIENTCONNS) THEN
		ClientDecOK = TRUE
	ELSE
		ClientDecOK = FALSE
		strcpy(ADR(Kanlink.ErrorString),"Declaration of HLKANLINK_MAX_CLIENTCONNS not large enough")
	ENDIF

	IF 	ServerDecOK AND ClientDecOK THEN

		;Server init
		IF Kanlink.Server.Enable THEN
			LOOP n = 1 TO Kanlink.Server.MaxConns DO
				;Build strings to pass to variable names, only required in a loop as index number changes.
				itoa(n,ADR(sn))	; put n into string
				strcpy(ADR(sReq),"PT100[");build string for variable name (request)
				strcat(ADR(sReq),ADR(sn))
				strcat(ADR(sReq),"].Req")
				strcpy(ADR(sResp),"PT100[");;build string for variable name (response)
				strcat(ADR(sResp),ADR(sn))
				strcat(ADR(sResp),"].Resp")
				IF Kanlink.Server.IP[n].AdvMode THEN
					IFhlKanLink.Parameter.Server[n].Adr = 0;
					IFhlKanLink.Parameter.Server[n].Area = 0
					IFhlKanLink.Parameter.Server[n].AdvMode := TRUE;
					strcpy(ADR(IFhlKanLink.Parameter.Server[n].AdrAdvMode),ADR(Kanlink.Server.IP[n].AdrAdvMode));
				ELSE
					IFhlKanLink.Parameter.Server[n].Adr = Kanlink.Server.IP[n].Adr ; Populate these arrays .
					IFhlKanLink.Parameter.Server[n].Area = Kanlink.Server.IP[n].Area
				ENDIF
				IFhlKanLink.Parameter.Server[n].Cmd = 1000 ; cmd from the server are always even
				IFhlKanLink.Parameter.Server[n].CmdOpt = Kanlink.Server.IP[n].CmdOpt
				IFhlKanLink.Parameter.Server[n].TimeOut = 1000 ;ms
				strcpy(ADR(IFhlKanLink.Parameter.Server[n].Name),"PT100") ; Diags Only
				strcpy(ADR(IFhlKanLink.Parameter.Server[n].sReq),ADR(sReq));"zzKanLink:PT100[0].Req")
				strcpy(ADR(IFhlKanLink.Parameter.Server[n].sResp),ADR(sResp));"zzKanLink:PT100[0].Resp")
			ENDLOOP
		ENDIF
		;Client Init
		IF Kanlink.Client.Enable THEN
			LOOP n = 1 TO Kanlink.Client.MaxConns DO
				itoa(n,ADR(sn))	; put n into string
				strcpy(ADR(sReq),"PTResp[");build string for variable name (request)
				strcat(ADR(sReq),ADR(sn))
				strcat(ADR(sReq),"].Req")
				strcpy(ADR(sResp),"PTResp[");;build string for variable name (response)
				strcat(ADR(sResp),ADR(sn))
				strcat(ADR(sResp),"].Resp")

				IF Kanlink.Client.IP[n].AdvMode THEN
					IFhlKanLink.Parameter.Client[n].Adr = 0;
					IFhlKanLink.Parameter.Client[n].Area = 0
					IFhlKanLink.Parameter.Client[n].AdvMode := TRUE;
					strcpy(ADR(IFhlKanLink.Parameter.Client[n].AdrAdvMode),ADR(Kanlink.Client.IP[n].AdrAdvMode));
				ELSE
					IFhlKanLink.Parameter.Client[n].Adr = Kanlink.Client.IP[n].Adr ; Populate these arrays .
					IFhlKanLink.Parameter.Client[n].Area = Kanlink.Client.IP[n].Area
				ENDIF
				IFhlKanLink.Parameter.Client[n].Cmd = 1000
				IFhlKanLink.Parameter.Client[n].CmdOpt = Kanlink.Client.IP[n].CmdOpt
				IFhlKanLink.Parameter.Client[n].CycleTime = 1000;ms
				strcpy(ADR(IFhlKanLink.Parameter.Client[n].Name),"PTResp")
				strcpy(ADR(IFhlKanLink.Parameter.Client[n].sReq),ADR(sReq))
				strcpy(ADR(IFhlKanLink.Parameter.Client[n].sResp),ADR(sResp))
			ENDLOOP
		ENDIF
		;Overview Server init
		;STOverResp[0] //Server sends batch data...
		IF Kanlink.OverviewServer.Enable THEN
			LOOP n = 1 TO Kanlink.OverviewServer.MaxConns DO
				;Build strings to pass to variable names, only required in a loop as index number changes.
				itoa(n,ADR(sn))	; put n into string
				strcpy(ADR(sReq),"STOverResp[");build string for variable name (request)
				strcat(ADR(sReq),ADR(sn))
				strcat(ADR(sReq),"].Req")
				strcpy(ADR(sResp),"STOverResp[");;build string for variable name (response)
				strcat(ADR(sResp),ADR(sn))
				strcat(ADR(sResp),"].Resp")

				Index = n + Kanlink.Server.MaxConns
				Kanlink.OverviewServer.IndexOffset = Kanlink.Server.MaxConns
				IF Kanlink.OverviewServer.IP[n].AdvMode THEN
					IFhlKanLink.Parameter.Server[Index].Adr = 0;
					IFhlKanLink.Parameter.Server[Index].Area = 0
					IFhlKanLink.Parameter.Server[Index].AdvMode := TRUE;
					strcpy(ADR(IFhlKanLink.Parameter.Server[Index].AdrAdvMode),ADR(Kanlink.OverviewServer.IP[n].AdrAdvMode));
				ELSE
					IFhlKanLink.Parameter.Server[Index].Adr = Kanlink.OverviewServer.IP[n].Adr ; Populate these arrays .
					IFhlKanLink.Parameter.Server[Index].Area = Kanlink.OverviewServer.IP[n].Area
				ENDIF

				IFhlKanLink.Parameter.Server[Index].Cmd = 1002 ;Batch Info Command
				IFhlKanLink.Parameter.Server[Index].CmdOpt = Kanlink.OverviewServer.IP[n].CmdOpt
				IFhlKanLink.Parameter.Server[Index].TimeOut = 1000 ;ms
				strcpy(ADR(IFhlKanLink.Parameter.Server[Index].Name),"STOverResp") ; Diags Only
				strcpy(ADR(IFhlKanLink.Parameter.Server[Index].sReq),ADR(sReq));"zzKanLink:STOverReq[0].Req")
				strcpy(ADR(IFhlKanLink.Parameter.Server[Index].sResp),ADR(sResp));"zzKanLink:STOverReq[0].Resp")

			ENDLOOP
		ENDIF

		;Kanlink OverView Client
		;STOverReq[0]// Client recieves batch data
		IF Kanlink.OverviewClient.Enable THEN
			LOOP n = 1 TO Kanlink.OverviewClient.MaxConns DO
				;Build strings to pass to variable names, only required in a loop as index number changes.
				itoa(n,ADR(sn))	; put n into string
				strcpy(ADR(sReq),"STOverReq[");build string for variable name (request)
				strcat(ADR(sReq),ADR(sn))
				strcat(ADR(sReq),"].Req")
				strcpy(ADR(sResp),"STOverReq[");;build string for variable name (response)
				strcat(ADR(sResp),ADR(sn))
				strcat(ADR(sResp),"].Resp")
				Index = n + Kanlink.Client.MaxConns
				Kanlink.OverviewClient.IndexOffset = Kanlink.Client.MaxConns

				IF Kanlink.OverviewClient.IP[n].AdvMode THEN
					IFhlKanLink.Parameter.Client[Index].Adr = 0;
					IFhlKanLink.Parameter.Client[Index].Area = 0
					IFhlKanLink.Parameter.Client[Index].AdvMode := TRUE;
					strcpy(ADR(IFhlKanLink.Parameter.Server[Index].AdrAdvMode),ADR(Kanlink.OverviewClient.IP[n].AdrAdvMode));
				ELSE
					IFhlKanLink.Parameter.Client[Index].Adr = Kanlink.OverviewClient.IP[n].Adr ; Populate these arrays .
					IFhlKanLink.Parameter.Client[Index].Area = Kanlink.OverviewClient.IP[n].Area
				ENDIF

				IFhlKanLink.Parameter.Client[Index].Cmd = 1002 ;Batch Info Command
				IFhlKanLink.Parameter.Client[Index].CmdOpt = Kanlink.OverviewClient.IP[n].CmdOpt
				IFhlKanLink.Parameter.Client[Index].CycleTime = 1000 ;ms
				strcpy(ADR(IFhlKanLink.Parameter.Client[Index].Name),"STOverReq") ; Diags Only
				strcpy(ADR(IFhlKanLink.Parameter.Client[Index].sReq),ADR(sReq));"zzKanLink:STOverResp[0].Req")
				strcpy(ADR(IFhlKanLink.Parameter.Client[Index].sResp),ADR(sResp));"zzKanLink:STOverResp[0].Resp")
			ENDLOOP
		ENDIF

		IFhlKanLink.in.xRestart = TRUE
		IFmnParam.Out.xParamOK = TRUE
		init = TRUE
		PT100 ; Variable that writes to the PT+ (Server)
		PTResp ; Variable that reads from PT+ (Client)
		STOverReq ;Variable used for the overview client
		STOverResp;Variable used for the overview server
	ENDIF//Server,client size OK
ENDIF//INIT

END_PROGRAM
```

### Program Logical/KanLink_A19/Kan_Driver (IEC, version 1.20.0) - *Kanlink Driver Server and Client

#### Kan_Driver.ab - Implementation code
```automation-basic
(********************************************************************
 * COPYRIGHT -- HP
 ********************************************************************
 * Program: Kan_Driver
 * File: Kan_Driver.ab
 * Author: treamsbottom
 * Created: September 07, 2012
 ********************************************************************
 * Implementation of program Kan_Driver
 ********************************************************************)
;----------------------------------------------------------------------------------------------------------------;
;-----21-1-2013..TR..Version A6 - First TestedVersion - Note 2 Specials in overview clien to run with Shuttle
;-----28-1-2013..TR..Version A7 - Remove Specials..Add option to send program and category number & Batch number.
;-----20-5-2014..TR..Version A12 - Fix ValidCat on DataValid
;-----09-01-2015..TR..Version A14 - Add Batching control
;-----02-08-2016 ..TR..Version A17 - Add Syncronous loading to Server Cmd 1000.. Use CAN[x].Transfer to watch for permission to unload.
;-----03-03-2017..TR.Version A18 - Add "Advanced Connection Mode"
;-----07-06-2017 ..TR..Version A19 - Fix issues with sending empty bag date-- Remove reference to CAN[].Category -- Read all information from bag for consistency.
;-----24-07-2018 ..TR -- Versioning Stopped Issues now tracked in GIT.
;-----------------------------------------------------------------------------------------------------------------

PROGRAM _CYCLIC
;Monitor State of supertrack (only send basic states now).
IF (Kanlink.Server.Enable OR Kanlink.Client.Enable OR Kanlink.OverviewClient.Enable OR Kanlink.OverviewServer.Enable) THEN
	IF Std.HaltSys THEN
		SuperTrackState = KG_MACHINESTATE_EMERGENCYSTOP
	ELSE
		SuperTrackState = KG_MACHINESTATE_AUTOMATIC_RUN
	ENDIF
ENDIF
;--------------------------------------------------Kanlink Server Communication-----------------------------------------------------------------
IF Kanlink.Server.Enable THEN
	;Populate Batch Data
	LOOP n = 1 TO Kanlink.Server.MaxConns  DO
		IF (Kanlink.Server.IP[n].Adr > 0) THEN
			LOOP Index = 1 TO 6 DO ; Loop through each bag buffer
				BagNumber = Kanlink.Server.BagNum[n].BagNums[Index]
				CANOffset = (Kanlink.Server.CANOffset - 1)
				IF (Bag[BagNumber].Prg > 0) AND (Bag[BagNumber].Prg <= Std.MaxProg)  THEN
					GetTimeStamp.enable = 1
					GetTimeStamp FUB DTGetTime()
					Batch[n].BatchData[Index].dtTimeStamp = GetTimeStamp.DT1
					;Make a string out OF CAT AND CUS
					length = itoa(Bag[BagNumber].Prg,ADR(myProgramString))
					length = itoa(Bag[BagNumber].Cat,ADR(myCategoryString));
					length = itoa(Bag[BagNumber].Cus,ADR(myCustomerString));

					;copy Bag Data to KanLink Bag data type
					IF Kanlink.GlobalSettings.TransferProgramCode THEN
						Batch[n].BatchData[Index].sCategory = myProgramString
						length = memcpy(ADR(Batch[n].BatchData[Index].bCustom),ADR(myCategoryString),12)
					ELSE IF Kanlink.GlobalSettings.TransferProgin_bCustom THEN
						Batch[n].BatchData[Index].sCategory = myCategoryString
						length = memcpy(ADR(Batch[n].BatchData[Index].bCustom),ADR(myProgramString),12)
					ELSE
						Batch[n].BatchData[Index].sCategory = myCategoryString
					ENDIF
					IF Kanlink.GlobalSettings.UseBatchCode THEN
						IF Kanlink.GlobalSettings.BatchCodeTyp = BatchTyp_UDINT THEN
							;length = itoa(Bag[BagNumber].Mis,ADR(Batch[n].BatchData[Index].bBatchNo)) ; Convert to string
							length = memcpy(ADR(Batch[n].BatchData[Index].bBatchNo),ADR(Bag[BagNumber].Mis),4) ; Direct UDINT copy unreadble in KANLINK data.
						ELSE IF Kanlink.GlobalSettings.BatchCodeTyp = BatchTyp_16Byte THEN
							;Bag typ does not support this yet..
						ENDIF
					ELSE
						length = strcpy(ADR(Batch[n].BatchData[Index].bBatchNo),"")
					ENDIF
					Batch[n].BatchData[Index].bCntCustomers = 1
					Batch[n].BatchData[Index].wTotalWeight = CAN[n + CANOffset].Weight;Summary weight of all Part Customers in the Bag, normally 1
					;First Customer in the Bag

					IF (CAN[n+ CANOffset].Batch_QtyRemaining <= 1) THEN
						Batch[n].BatchData[Index].PartBatch[0].sCustomNo = myCustomerString
						Batch[n].BatchData[Index].PartBatch[0].wCustomWeight = Bag[BagNumber].Wgt
					ELSE
						Batch[n].BatchData[Index].bCntCustomers = USINT(CAN[n+ CANOffset].Batch_QtyRemaining)
						LOOP t = 0 TO 7 DO
							length = itoa(CAN[n + CANOffset].Batchpart[t].Customer,ADR(myCustomerString));
							Batch[n].BatchData[Index].PartBatch[t].sCustomNo = myCustomerString
							Batch[n].BatchData[Index].PartBatch[t].wCustomWeight = CAN[n + CANOffset].Batchpart[t].Wgt
						ENDLOOP
					ENDIF
				ELSE
					strcpy(ADR(myCategoryString),ADR(""));
					strcpy(ADR(myCustomerString),ADR(""))
					strcpy(ADR(myProgramString),ADR(""));
					Batch[n].BatchData[Index].bCntCustomers = 0
					Batch[n].BatchData[Index].sCategory = myCategoryString
					length = strcpy(ADR(Batch[n].BatchData[Index].bCustom),"")
					length = strcpy(ADR(Batch[n].BatchData[Index].bBatchNo),"")
					Batch[n].BatchData[Index].wTotalWeight = 0 ;Summaray weight of all Part Customers in the Bag, normally 1
					LOOP t = 0 TO 7 DO
						Batch[n].BatchData[Index].PartBatch[t].sCustomNo = myCustomerString
						Batch[n].BatchData[Index].PartBatch[t].wCustomWeight = 0
					ENDLOOP
				ENDIF
				PT100[n].Resp.BatchData = Batch[n].BatchData[1] ; Only send first bag over KANLINK
			ENDLOOP

			; Handshake Signal Convert CAN into the KANLINK protocol
			;ValidCat = 	strcmp(ADR(CAN[n + CANOffset].Category), "")
			BagNumber = Kanlink.Server.BagNum[n].BagNums[1];
			IF (Bag[BagNumber].Cat > 0)  AND (CAN[n + CANOffset].Category > 0) THEN
				PT100[n].Resp.xHsDataValid = TRUE;
			ELSE
				PT100[n].Resp.xHsDataValid = FALSE
				PT100[n].Resp.xHsUnloading = FALSE
			ENDIF

			IF CAN[n + CANOffset].BagReady THEN
				PT100[n].Resp.xHsReqForUnload = TRUE;
			ELSE
				PT100[n].Resp.xHsReqForUnload = FALSE;
			ENDIF

			CAN[n+CANOffset].DropLoad 		= PT100[n].Req.xHreadyForLoad;
			CAN[n+CANOffset].LoadDropped  	= PT100[n].Req.xHbatchReceived;
			PT100[n].Resp.wCntLoads = CAN[n + CANOffset].Batch_QtyRemaining

			IF CAN[n+CANOffset].DropLoad THEN
				PT100[n].Resp.xHsUnloading = TRUE
			ENDIF
			PT100[n].Resp.wState = SuperTrackState
			CAN[n+CANOffset].Live = IFhlKanLink.Server[n].out.xConnected
		;Syncronous Loading.
			IF PT100[n].Req.xHreqCtrlTransfer THEN
				//Syncronous loading. Only allow unload when bit .x.x.x. is on
				PT100[n].Resp.xHsTransferRunning := PT100[n].Req.xHwaitingForTransfer;
			ELSE
				//Always give permission to unload..
				PT100[n].Resp.xHsTransferRunning := 1;
			ENDIF;
			CAN[n+CANOffset].Transfer := PT100[n].Resp.xHsTransferRunning
		ENDIF
	ENDLOOP
ENDIF//ServerDriver
;--------------------------------------------------------Client Driver------------------------------------------------------------------
IF Kanlink.Client.Enable THEN
	LOOP n = 1 TO Kanlink.Client.MaxConns DO
		CANOffset = (Kanlink.Client.CANOffset - 1)
		;Give Machine Ready
		PTResp[n].Req.xHready = NOT Std.HaltSys
		PTResp[n].Req.xHcmdAutomatic = TRUE

		CAN[n + CANOffset].BagReady = PTResp[n].Resp.xHsReqForUnload
		;Give ready to load when Ready
		PTResp[n].Req.xHreadyForLoad = CAN[n + CANOffset].ReadyToLoad

		PTResp[n].Req.xHbatchReceived = CAN[n + CANOffset].LoadRecieved
		;Send supertrack state
		PTResp[n].Req.wHstate = SuperTrackState

		;Check for Data Valid and unloading start.	then copy data to CAN Variable
		UnloadingPulse[n].CLK = (PTResp[n].Resp.xHsUnloading AND PTResp[n].Resp.xHsDataValid)
		UnloadingPulse[n] FUB R_TRIG()
		IF UnloadingPulse[n].Q THEN
			IF Kanlink.GlobalSettings.TransferProgramCode THEN
				CAN[n + CANOffset].Program = USINT(atoi(ADR(PTResp[n].Resp.BatchData.sCategory)))
				CAN[n + CANOffset].Category = atoi(ADR(PTResp[n].Resp.BatchData.bCustom))
			ELSE IF Kanlink.GlobalSettings.TransferProgin_bCustom THEN
				CAN[n + CANOffset].Program = USINT(atoi(ADR(PTResp[n].Resp.BatchData.bCustom)))
				CAN[n + CANOffset].Category = atoi(ADR(PTResp[n].Resp.BatchData.sCategory))
			ELSE
				CAN[n + CANOffset].Category = atoi(ADR(PTResp[n].Resp.BatchData.sCategory))
			ENDIF
			CAN[n + CANOffset].Customer = atoi(ADR(PTResp[n].Resp.BatchData.PartBatch[0].sCustomNo))
			CAN[n + CANOffset].Weight = PTResp[n].Resp.BatchData.wTotalWeight
			IF Kanlink.GlobalSettings.UseBatchCode THEN
				IF Kanlink.GlobalSettings.BatchCodeTyp = BatchTyp_UDINT THEN
					length = memcpy(ADR(CAN[n + CANOffset].BatchID),ADR(PTResp[n].Resp.BatchData.bBatchNo),4)
				ELSE IF Kanlink.GlobalSettings.BatchCodeTyp = BatchTyp_16Byte THEN
					;Bag typ does not support this yet..
				ENDIF
			ELSE
				CAN[n + CANOffset].BatchID = 0
			ENDIF
		ENDIF

		CAN[n + CANOffset].Unloading =  PTResp[n].Resp.xHsUnloading
		UnloadingFinishPLS[n].CLK = PTResp[n].Resp.xHsUnloading
		UnloadingFinishPLS[n] FUB F_TRIG()

		CAN[n + CANOffset].UnloadFinished = UnloadingFinishPLS[n].Q
		;Can Live
		CAN[n+CANOffset].Live = IFhlKanLink.Client[n].out.xConnected
	ENDLOOP
ENDIF
;---------------------------------------------------------------------------------------------Overview Client----------------------------------------
IF Kanlink.OverviewClient.Enable THEN ; Collect data
;------------------------------------------Build Request---------------------------------------------------

	LOOP n = 1 TO Kanlink.OverviewClient.MaxConns DO

		IF (CANOffset > 0) THEN
			CANOffset = (Kanlink.OverviewClient.CANOffset - 1)
			CAN[n+CANOffset].Live = IFhlKanLink.Client[n+Kanlink.OverviewClient.IndexOffset].out.xConnected
			IF NOT CAN[n+CANOffset].Live THEN
				D[Kanlink.OverviewClient.StatusReg[n]] = 0
			ENDIF
		ELSE
			CANOffset = 0
		ENDIF;

		IF Kanlink.OverviewClient.InfoReq[n].wNoOfPosition[6] = 0 THEN ; do not multiplex data.
			STOverReq[n].Req.wCntPositions = Kanlink.OverviewClient.InfoReq[n].wCntPositions;Number of Bags requested
			DataOffset[n] = 0
		ELSE

			DataCount = 0
			LOOP x = 0 TO 5 DO
				IF (STOverReq[n].Req.wNoOfPosition[x] > 0) THEN
					DataCount = DataCount + 1
				ENDIF
				IF DataCount > 5 THEN
					DataCount = 6
				ENDIF
			ENDLOOP
			STOverReq[n].Req.wCntPositions = DataCount;Number of Bags requested
		ENDIF

		LOOP x = 0 TO 5 DO
			;datapositions requested
			EXITIF ((DataOffset[n] + x) > HLKANLINK_MAX_OVERVIEW_DATA)

			STOverReq[n].Req.wNoOfPosition[x] = Kanlink.OverviewClient.InfoReq[n].wNoOfPosition[x + DataOffset[n]]
				;-----------------------------------------------Read Data----------------------------------
			IF (STOverReq[n].Resp.wNoOfPositions[x] > 0) AND ((x <= STOverReq[n].Resp.wCntPositions) OR (STOverReq[n].Resp.wCntPositions = 0 )) THEN
				IF (Kanlink.OverviewClient.InfoResp[n].BagNum[x + DataOffset[n]] > 0) THEN
					IF Kanlink.OverviewClient.InfoReq[n].wNoOfPosition[x+DataOffset[n]] = STOverReq[n].Resp.wNoOfPositions[x] THEN
					//	D[Kanlink.OverviewClient.StatusReg[n]] = STOverReq[n].Resp.wMachineState
						BagIndex = Kanlink.OverviewClient.InfoResp[n].BagNum[x + DataOffset[n]]
						IF Kanlink.GlobalSettings.TransferProgramCode THEN
							Bag[BagIndex].Prg = USINT(atoi(ADR(STOverReq[n].Resp.BatchData[x].sCategory)))
							Bag[BagIndex].Cat = atoi(ADR(STOverReq[n].Resp.BatchData[x].bCustom))
						ELSE IF Kanlink.GlobalSettings.TransferProgin_bCustom THEN
							Bag[BagIndex].Prg = USINT(atoi(ADR(STOverReq[n].Resp.BatchData[x].bCustom)))
							Bag[BagIndex].Cat = atoi(ADR(STOverReq[n].Resp.BatchData[x].sCategory))
						ELSE
							Bag[BagIndex].Cat = atoi(ADR(STOverReq[n].Resp.BatchData[x].sCategory))
						ENDIF
						Bag[BagIndex].Cus = atoi(ADR(STOverReq[n].Resp.BatchData[x].PartBatch[0].sCustomNo)) ; Standard line of code..
						Bag[BagIndex].Wgt = STOverReq[n].Resp.BatchData[x].PartBatch[0].wCustomWeight
						IF Kanlink.GlobalSettings.UseBatchCode THEN
							IF Kanlink.GlobalSettings.BatchCodeTyp = BatchTyp_UDINT THEN
									length = memcpy(ADR(Bag[BagIndex].Mis),ADR(STOverReq[n].Resp.BatchData[x].bBatchNo),4)
								ELSE IF	Kanlink.GlobalSettings.BatchCodeTyp = BatchTyp_16Byte THEN
								;Not supported yet....
							ENDIF
						ELSE
							Bag[BagIndex].Mis = 0
						ENDIF
					ENDIF
				ENDIF
			ENDIF
		ENDLOOP
		IF STOverReq[n].Resp.wNoOfPositions[0] = Kanlink.OverviewClient.InfoReq[n].wNoOfPosition[DataOffset[n]] THEN
			DataOffset[n] = DataOffset[n] + 6
		ELSE IF Kanlink.OverviewClient.InfoReq[n].wNoOfPosition[DataOffset[n]] = 0 THEN
			DataOffset[n] = 0
		ENDIF
	ENDLOOP
ENDIF

;---------------------------------------------------------------------------------------------Overview Server----------------------------------------
IF Kanlink.OverviewServer.Enable THEN
	LOOP n = 1 TO Kanlink.OverviewServer.MaxConns DO
		IF (STOverResp[n].Req.wCntPositions <= 6) THEN
			IF (STOverResp[n].Req.wCntPositions = 0) OR (STOverResp[n].Req.wCntPositions = 6) THEN
				NoOfDataRequested = 5
			ELSE
				NoOfDataRequested = STOverResp[n].Req.wCntPositions
			ENDIF
			LOOP x = 0 TO 5 DO
				IF x <= NoOfDataRequested THEN
					BagIndex = STOverResp[n].Req.wNoOfPosition[x]

					//STOverResp[n].Resp.wMachineState = SuperTrackState
					STOverResp[n].Resp.wNoOfPositions[x] = BagIndex
					STOverResp[n].Resp.wCntPositions = 	STOverResp[n].Req.wCntPositions
					itoa(Bag[BagIndex].Prg,ADR(sProgram))
					itoa(Bag[BagIndex].Cat,ADR(sCategory))
					itoa(Bag[BagIndex].Cus,ADR(sCustomer))
					itoa(Bag[BagIndex].Mis,ADR(sBatchID))
					STOverResp[n].Resp.BatchData[x].dtTimeStamp = GetTimeStamp.DT1
					IF Kanlink.GlobalSettings.TransferProgramCode THEN
						strcpy(ADR(STOverResp[n].Resp.BatchData[x].sCategory),ADR(sProgram))
						strcpy(ADR(STOverResp[n].Resp.BatchData[x].bCustom),ADR(sCategory))
					ELSE IF Kanlink.GlobalSettings.TransferProgin_bCustom THEN
						strcpy(ADR(STOverResp[n].Resp.BatchData[x].sCategory),ADR(sCategory))
						strcpy(ADR(STOverResp[n].Resp.BatchData[x].bCustom),ADR(sProgram))
					ELSE
						strcpy(ADR(STOverResp[n].Resp.BatchData[x].sCategory),ADR(sCategory))
					ENDIF
					IF Kanlink.GlobalSettings.UseBatchCode THEN
						IF Kanlink.GlobalSettings.BatchCodeTyp = BatchTyp_UDINT THEN
							length = memcpy(ADR(STOverResp[n].Resp.BatchData[x].bBatchNo),ADR(Bag[BagIndex].Mis),4)
						ELSE IF Kanlink.GlobalSettings.BatchCodeTyp = BatchTyp_UDINT THEN
							strcpy(ADR(STOverResp[n].Resp.BatchData[x].bBatchNo),ADR(sBatchID))
						ENDIF
					ELSE
						strcpy(ADR(STOverResp[n].Resp.BatchData[x].bBatchNo),"")
					ENDIF
					strcpy(ADR(STOverResp[n].Resp.BatchData[x].PartBatch[0].sCustomNo),ADR(sCustomer))
					STOverResp[n].Resp.BatchData[x].PartBatch[0].wCustomWeight = Bag[BagIndex].Wgt
				ELSE
					STOverResp[n].Resp.wNoOfPositions[x] = 0
					STOverResp[n].Resp.BatchData[x].dtTimeStamp = 0
					strcpy(ADR(STOverResp[n].Resp.BatchData[x].sCategory),"")
					strcpy(ADR(STOverResp[n].Resp.BatchData[x].bCustom),"")
					strcpy(ADR(STOverResp[n].Resp.BatchData[x].bBatchNo),"")
					strcpy(ADR(STOverResp[n].Resp.BatchData[x].PartBatch[0].sCustomNo),"")
					STOverResp[n].Resp.BatchData[x].PartBatch[0].wCustomWeight = 0
				ENDIF
			ENDLOOP
		ENDIF
	ENDLOOP
ENDIF

END_PROGRAM
```

#### Kan_Driver.var - Local variables
```iecst
(********************************************************************
 * COPYRIGHT -- HP
 ********************************************************************
 * Program: Kan_Driver
 * File: Kan_Driver.var
 * Author: treamsbottom
 * Created: September 07, 2012
 ********************************************************************
 * Local variables of program Kan_Driver
 ********************************************************************)
VAR
	n : UINT;
	Index : UINT;
	BagNumber : UINT;
	CANOffset : UINT;
	GetTimeStamp : DTGetTime;
	length : UDINT;
	ValidCat : UDINT;
	myCategoryString : STRING[11];
	myCustomerString : STRING[11];
	UnloadingPulse : ARRAY[0..HLKANLINK_MAX_CLIENTCONNS] OF R_TRIG;
	UnloadingFinishPLS : ARRAY[0..HLKANLINK_MAX_CLIENTCONNS] OF F_TRIG;
	SuperTrackState : USINT;
	x : UINT;
	BagIndex : UINT;
	sCustomer : STRING[11];
	sCategory : STRING[11];
	sBatchID : STRING[16];
	NoOfDataRequested : UINT;
	DataOffset : ARRAY[0..HLKANLINK_MAX_CLIENTCONNS] OF UINT;
	DataCount : UINT;
	str_n : STRING[2];
	myProgramString : STRING[11];
	sProgram : STRING[11];
	t : UINT;
END_VAR
```

### Package Logical/KanLink_A19/KGFramework - Standard-Packages

### Package Logical/KanLink_A19/KGFramework/Pkg_KGStandard - Kannegiesser Standards

### Library Logical/KanLink_A19/KGFramework/Pkg_KGStandard/KGstdLib (IEC) - Kannegiesser Hilfsfunktionen
Depends on: astime, AsIODiag, Ethernet, AsBrStr, DataObj, AsArLog

#### kgGetEthPort.st - Returns the CPUs ethernet port as string
```iecst
(********************************************************************
 * COPYRIGHT -- Microsoft
 ********************************************************************
 * Library: Netlink
 * File: GetEthPort.st
 * Author: hunholz
 * Created: June 30, 2011
 ********************************************************************
 * Implementation of library Netlink
 ********************************************************************)

(* Returns the CPUs ethernet port as string *)
FUNCTION_BLOCK kgGetEthPort

	IF enable THEN

		IF adrIF <= 16#3FFF THEN

			_bStep := 10;
			status := KG_ERR_GETETHPORT_ADRIF;
			RETURN;

		END_IF

		_xReady := FALSE;

		REPEAT

			CASE (_bStep) OF

				10:
				// Create Info
					DiagCreateInfo_CPU(enable := TRUE, infoKind := asdiagPLUGGED);

					status := DiagCreateInfo_CPU.status;

					IF (status = ERR_OK) THEN
			  			_bStep := 12;
					END_IF;

				12:
					// Get Info
					DiagGetNumInfo_CPU(enable := TRUE,
											ident := DiagCreateInfo_CPU.ident,
											index := 0,
											infoCode := asdiagPLUGGED_MODNO);

					status := DiagGetNumInfo_CPU.status;

					IF (status = ERR_OK) THEN

						CASE DiagGetNumInfo_CPU.value OF

							KG_CPU_X20CP1484, KG_CPU_X20CP1484_1, KG_CPU_X20CP3484_1, KG_CPU_X20CP1486, KG_CPU_X20CP3486, KG_CPU_X20CP3585, KG_CPU_X20CP1584,KG_CPU_X20CP1586, KG_CPU_X20CP3484:
								brsstrcpy(adrIF, ADR('IF2'));

							KG_CPU_PP420_1043_75, KG_CPU_CTT_11, KG_CPU_PP65_0571_P74, KG_CPU_PCT_04, KG_CPU_PCT_03:
								brsstrcpy(adrIF, ADR('IF5'));

							ELSE	// keinen gültigen B&R ID-Code gefunden
								brsstrcpy(adrIF, ADR('ERR'));
								status := KG_ERR_GETETHPORT_IFSTRING;

						END_CASE

						_bStep := 14;

					ELSIF (status <> ERR_FUB_BUSY) THEN
						_bStep := 10;
					END_IF;

				14:
					// Write string to variable

					DiagDisposeInfo_CPU(enable := TRUE, ident := DiagCreateInfo_CPU.ident);

					status := DiagDisposeInfo_CPU.status;

					_xReady := (status = ERR_OK);

					IF (status <> ERR_FUB_BUSY) THEN

						_bStep := 10;
						DiagCreateInfo_CPU(enable := FALSE);
						DiagDisposeInfo_CPU(enable := FALSE);
						DiagGetNumInfo_CPU(enable := FALSE);

					END_IF;

				ELSE

					_bStep := 10;
					status := ERR_FUB_BUSY;

			END_CASE;

			UNTIL

			status <> ERR_OK OR _xReady

		END_REPEAT

	ELSE

		status := ERR_FUB_ENABLE_FALSE;
		_bStep := 10;

	END_IF

END_FUNCTION_BLOCK
```


- Program Logical/KanLink_A19/KGFramework/Pkg_mnSystem/mnSystem (IEC) - Systemtask für Versionierung (no source held here)

- Program Logical/KanLink_A19/KGFramework/Pkg_mnEth/mnEth (IEC) - Ethernetmanager (no source held here)

- Program Logical/KanLink_A19/KGFramework/Pkg_mnCnt/mnCnt (IEC) - Counter Manager (no source held here)

- Program Logical/KanLink_A19/KGFramework/Pkg_mnMsg/mnMsg (IEC) - Meldungsmanager (no source held here)

- Library Logical/KanLink_A19/KGFramework/Pkg_mnMsg/KGlibMsg (IEC) - A new source library (no source held here)

### Package Logical/KanLink_A19/KGFramework/Pkg_mnParam - Parameter-Manager

- Program Logical/KanLink_A19/KGFramework/Pkg_mnParam/mnParam (IEC) - Parameter Manager (no source held here)

### Library Logical/KanLink_A19/KGFramework/Pkg_mnParam/mnParamLib (IEC)
Depends on: astime


- Program Logical/KanLink_A19/KGFramework/Pkg_mnTxt/mnTxt (IEC) - Text-Manager (no source held here)

- Program Logical/KanLink_A19/KGFramework/Pkg_hlDFII/hlDFII (IEC) - Statemachine zur Abfrage einer SQL-Datenbank (no source held here)

- Program Logical/KanLink_A19/KGFramework/Pkg_mnTest/mnTest (IEC) - Testadapter (no source held here)

- Program Logical/KanLink_A19/KGFramework/Pkg_svCPCache/svCPCache (IEC) - Category-Program-Cache (no source held here)

### Program Logical/KanLink_A19/KGFramework/Pkg_hlKanLink/hlKanLink (IEC) - Kanlink Task

#### KanLink.var - Local variables
```iecst
(********************************************************************
 * COPYRIGHT -- Herbert Kannegiesser GmbH
 ********************************************************************
 * Program: WetLink
 * File: WetLink.var
 * Author: stahlhut
 * Created: December 23, 2011
 ********************************************************************
 * Local variables of program WetLink
 ********************************************************************)
VAR
	_xIdxFound : BOOL;
	_ptrIndex : REFERENCE TO KL_ServerListe_typ;
	_i : UINT;
	_iCltRespCnt : INT;
	_xCltFound : BOOL;
	_xInitOK : BOOL;
	_kgArLogWrite : kgArLogWrite;
	_AsArLogCreate : AsArLogCreate;
	_AsArLogGetInfo : AsArLogGetInfo;
	_wPtrRBwrite : UINT;
	_wPtrRBread : UINT;
	_wPtrRBstart : UINT;
	_kgRBcreateKanLinklog : kgRBcreate;
	_wPtrRBloc : UINT;
	_xRBReady : BOOL;
	_InsertRB : kgRBinsert;
	_ReadRB : kgRBread;
	_LogEntry : ErrLog_typ;
	_LogEntryIn : ErrLog_typ;
	_wLogStep : UINT;
	_MemPartCreate : AsMemPartCreate;
	_lTempMemIdent : UDINT;
	_lMemIdent : UDINT;
	_MemAlloc : AsMemPartAllocClear;
END_VAR
VAR RETAIN
	_iLastCltIdx : UINT;
END_VAR
VAR
	_dClient : REFERENCE TO KL_ClientListe_typ;
	_xAdrErr : BOOL;
	_iIdxFound : INT;
	_xAdrOK : BOOL;
	WL_ErrorNr : UINT;
	KL_SaveConfDO_0 : KL_SaveConfDO;
	_xSaveConfig : BOOL;
	_iLastServerIdx : UINT;
	_xServerFound : BOOL;
	_dSrvIf : REFERENCE TO IF_Server_typ;
	_dCltIf : REFERENCE TO IF_Client_typ;
	_ifDummy : IF_Client_typ;
	_xSendNow : BOOL;
	Kanlink : KanLink_FB;
	_sPkgName : STRING[11];
	_VerStruc : MoVerStruc_typ;
	_lAdr : UDINT;
	_lLen : UDINT;
	_wStatus : UINT;
	_MemAllocTemp : AsMemPartAllocClear;
END_VAR
VAR CONSTANT
	_HLKANLINK_IDX_STRUCDEF_RESP_0 : UINT := 1;
END_VAR
VAR
	_lPtrStrucDef : ARRAY[0..5] OF UDINT;
	_lPtrStrucLen : ARRAY[0..5] OF UDINT;
	_MemFreeTemp : AsMemPartFree;
	_wDebIdx : UINT;
END_VAR
VAR CONSTANT
	_HLKANLINK_MAX_IDX_DEFSTRUC : UINT := 5;
END_VAR
VAR
	_sDebString : REFERENCE TO STRING[31];
	_wDebOffset : UINT;
	_sName : STRING[80];
	_state : USINT;
	_tcnr : SINT;
	_wClt : UINT;
	_wSrv : UINT;
END_VAR
```

#### KanLinkCyclic.st - Cyclic code
```iecst
(********************************************************************
 * COPYRIGHT -- Herbert Kannegiesser GmbH
 ********************************************************************
 * Program: KanLink
 * File: KanLinkCyclic.st
 * Author: stahlhut
 * Created: December 23, 2011
 ********************************************************************
 * Implementation of program WetLink
 ********************************************************************)

(*

	Falls ohne Framework gearbeitet werden soll in den Eigenschaften der Task hlKanLink (Config. View Cpu.sw)
	im Tab. Compiler im Feld "Additional build options:" -D HLKANLINK_AUTONOM  eintragen
	Dazu das Package KanLinkAutonom importieren

*)

PROGRAM _CYCLIC

// Struktur für Visualisierung füllen

IFhlKL_Visu.out.iCycleTime := Kanlink._iCycleTime;
IFhlKL_Visu.out.step := Kanlink.Step;
IFhlKL_Visu.out.udNetId := Kanlink.udNetID;
IFhlKL_Visu.out.udpOpenStatus := Kanlink.udp.open.status;
IFhlKL_Visu.out.udpRecStatus := Kanlink.udp.rec.status;
IFhlKL_Visu.out.udpSendStatus := Kanlink.udp.send.status;
_wClt := LIMIT(0,IFhlKL_Visu.in.iCltNr,HLKANLINK_MAX_CLIENTCONNS);
_wSrv := LIMIT(0,IFhlKL_Visu.in.iServerNr,HLKANLINK_MAX_SERVERCONNS);
IFhlKL_Visu.out.client := Kanlink.ClientListe[_wClt];
IFhlKL_Visu.out.server := Kanlink.ServerListe[_wSrv];

// Commando von der Visu verarbeiten
// Commando nur setzen wenn CmdResp = 0
// aufrufer muss nach ausführung cmdNr wieder auf 0 setzen!
IF IFhlKL_Visu.in.cmdNr <> IFhlKL_Visu.out.cmdResp THEN
	CASE IFhlKL_Visu.in.cmdNr OF
		0: IFhlKL_Visu.out.cmdResp := 0;
		1: // Neustart
			IFhlKL_Visu.out.cmdResp := 1;
			Kanlink.Step := 1;
		2: // Neustart mit lastId = 1
			Kanlink._uiLastId := 1;
			IFhlKL_Visu.out.cmdResp := 1;
			Kanlink.Step := 2;
		ELSE
			// unbekanntes Commando
			IFhlKL_Visu.out.cmdResp := 16#7FFF;

	END_CASE;
END_IF;

#ifndef HLKANLINK_AUTONOM // Logging nur mit kg-Framework

	// ===========================
	// Logging
	// ===========================

	IF _xRBReady THEN

		CASE _wLogStep OF

			0:
				_ReadRB(wPtrRead := _wPtrRBread, wPtrStart := _wPtrRBstart, wPtrWrite := _wPtrRBwrite);

				IF _ReadRB.wStatus = ERR_OK THEN

					CASE _LogEntry.wErrorNo OF

						0:
							_kgArLogWrite.text := 'OK';

						HLKANLINK_MSG_NO_STRUCDEF:

							_kgArLogWrite.text := 'Create Strucdefinition failed : {##AttrVar1} / {##AttrVar2}';
							_kgArLogWrite.var1 := _LogEntry.lAttr1;

						ELSE

							_kgArLogWrite.text := UINT_TO_STRING(_LogEntry.wErrorNo);
							_kgArLogWrite.text := CONCAT(_kgArLogWrite.text, ' : {##AttrVar1} / {##AttrVar2}');
							_kgArLogWrite.var1 := _LogEntry.lAttr1;
							_kgArLogWrite.var2 := _LogEntry.lAttr2;

					END_CASE

					_wLogStep := 1;

				END_IF

			1:
				_kgArLogWrite();

				IF _kgArLogWrite.status <> ERR_FUB_BUSY THEN

					_wLogStep := 0;

				END_IF

		END_CASE

	END_IF

	IF _wDebIdx >= 0 AND _wDebIdx <= _HLKANLINK_MAX_IDX_DEFSTRUC THEN

		IF _lPtrStrucDef[_wDebIdx] > 0 THEN

			_sDebString ACCESS _lPtrStrucDef[_wDebIdx] + _wDebOffset;

		END_IF

	END_IF

#endif

	// =======================================================================

	IF _xInitOK THEN

		IF _xSaveConfig THEN
			KL_SaveConfDO_0(adrName :=ADR('KL_Conf') , adrDaten := ADR(IFhlKanLink.Parameter), len := SIZEOF( IFhlKanLink.Parameter));
			IF KL_SaveConfDO_0.status <> ERR_FUB_BUSY THEN // fertig
				_xSaveConfig := FALSE;
			END_IF;
		END_IF;

		IF EDGEPOS(IFhlKanLink.in.xRun ) THEN
			IF Kanlink.Step = 0 THEN
				Kanlink.Step := 1;
			END_IF;
		END_IF;
		IF EDGENEG(IFhlKanLink.in.xRun) THEN // stoppen
			IF Kanlink.Step <> 0 THEN
				Kanlink.Step := 20;
			END_IF;
		END_IF;

		IF IFhlKanLink.in.xRestart THEN
			Kanlink.Step := 1;
			IFhlKanLink.in.xRestart := 0;
		END_IF;

		IFhlKanLink.xError := (Kanlink.Step = 200);

		CASE Kanlink.Step OF

			0: //nix tun

			100: // Error nr in Logger eintragen

				Kanlink.Step := 200;

			200: // Auf User warten

			1: // init

				Kanlink.KLLib_Init_0(enable := 1, adrServer := ADR(Kanlink),adrInterface := ADR(IFhlKanLink));
				IF Kanlink.KLLib_Init_0.status = ERR_OK THEN
					Kanlink.Step := 10;
				ELSIF Kanlink.KLLib_Init_0.status <> ERR_FUB_BUSY THEN // fehler
					WL_ErrorNr := 10;
					Kanlink.Step := 100;

					IF _xRBReady THEN

						_LogEntryIn.wErrorNo := 10;
						_InsertRB(wPtrStart := _wPtrRBstart, wPtrRead := _wPtrRBread, wPtrWrite := _wPtrRBwrite);

					END_IF

				END_IF;

			10: // Kanlink Run

			20: // Kanlink schliessen

				Kanlink.udp.close.enable := 1;
				Kanlink.udp.close.ident := Kanlink._uiLastId;
				Kanlink.udp.close;
				IF Kanlink.udp.close.status = 0 THEN
					Kanlink.Step := 0;
				ELSIF Kanlink.udp.close.status = ERR_FUB_BUSY THEN

				ELSE
					Kanlink.Step := 100;
				END_IF;

		END_CASE;

		// hier beenden wenn zyklus nicht erlaubt
		IF  Kanlink.Step <> 10 THEN
			RETURN;
		END_IF;

		Kanlink;

		// falls Kanlink nix zu tun hat, hier beenden
		IF Kanlink.xReturn THEN
			RETURN;
		END_IF;

		// ------------------------------------------------------------------
		// Falls ein Request eines Clients aufgelaufen ist

		IF Kanlink._xGetServerReq THEN  // Req eines Clients angenommen, bearbeiten

			actGetServerReq;

			Kanlink._xGetServerReq := FALSE;
			Kanlink.udp.rec.enable := 1;

			RETURN;  // Daten sind versendet. Also Ende.

		END_IF;

		// ------------------------------------------------------------------------------
		// falls Response von einem Request kommt:

		IF Kanlink._xGetClientResp THEN // Response auf ClientReq angekommen
			actResponse;

		END_IF;

		// ------------------------------------------------------------------------------
		// Überprüfen ob per Hand bearbeitete Requests versendet werden müssen..

		IF  Kanlink.udp.send.enable = 0 THEN
			_xServerFound := 0;

			FOR _i:=0 TO HLKANLINK_MAX_SERVERCONNS  DO
				_ptrIndex ACCESS ADR(Kanlink.ServerListe[_iLastServerIdx]);
				_dSrvIf ACCESS _ptrIndex.adrInterface;
				IF (_ptrIndex.xReqManually AND (_dSrvIf.iState = 2)) THEN
					_xServerFound := 1;

					_iLastServerIdx := _iLastServerIdx + 1; // testen
					IF _iLastCltIdx > HLKANLINK_MAX_SERVERCONNS THEN
						_iLastServerIdx := 0;
					END_IF;
					EXIT;
					END_IF;
					_iLastServerIdx := _iLastServerIdx + 1; // testen
					IF _iLastServerIdx > HLKANLINK_MAX_SERVERCONNS THEN
					_iLastServerIdx := 0;
				END_IF;

			END_FOR;

			IF _xServerFound THEN
				Kanlink.ServerData.HeaderV1Send.Command := _ptrIndex.Cmd + 1;
				Kanlink.ServerData.HeaderV1Send.dataFormat := 5;
				Kanlink.ServerData.HeaderV1Send.Length := UDINT_TO_UINT( _ptrIndex.RespLength);
				Kanlink.ServerData.HeaderV1Send.ReqID := _ptrIndex.iReqID;
				Kanlink.ServerData.HeaderV1Send.CmdNr := _ptrIndex.CmdOpt AND 16#000F;
				_ptrIndex.iConnectionTimer := 0;
				KLLib_SendData(ADR(Kanlink),_ptrIndex.AdrDataResp,_ptrIndex.RespLength,ADR(_ptrIndex.sClientIPAdr));
				_dSrvIf.iState := 0;
				RETURN;
			END_IF;
		END_IF;

		IF Kanlink._xSendClient THEN  // hier den Clienten bearbeiten

			_xCltFound := FALSE;

			FOR _i:=0 TO HLKANLINK_MAX_CLIENTCONNS  DO
				_dClient ACCESS ADR(Kanlink.ClientListe[_iLastCltIdx]);
				IF _dClient.adrInterface <> 0 THEN
					_dCltIf ACCESS _dClient.adrInterface;
				ELSE
					_dCltIf ACCESS ADR(_ifDummy);
				END_IF;
					// gefunden wenn kein ReqPend, Commando <> 0 todo gültige Adresse etc...
				IF _dClient.iCycleTime = 0 THEN
					_xSendNow := (_dCltIf.iState = 1) OR (_dCltIf.iState = 4) ; // falls angetickt oder timeout
				ELSE
					_xSendNow := (_dClient.iCycleWait > _dClient.iCycleTime);
				END_IF;
				IF 	(NOT _dClient.xReqPending) AND (_dClient.Cmd <> 0) AND  _dClient.xActiv AND (_xSendNow)   THEN
		  			_xCltFound := TRUE;
					_iLastCltIdx := _iLastCltIdx + 1; // testen
					IF _iLastCltIdx > HLKANLINK_MAX_CLIENTCONNS THEN
			  			_iLastCltIdx := 0;
					END_IF;
					EXIT;
				END_IF;

				_iLastCltIdx := _iLastCltIdx + 1; // testen
				IF _iLastCltIdx > HLKANLINK_MAX_CLIENTCONNS THEN
		  			_iLastCltIdx := 0;
				END_IF;

			END_FOR;

			IF NOT _xCltFound THEN
				Kanlink._xSendClient := FALSE;
				RETURN;

			ELSE

				// Client gefunden
				_dClient.iCnt := _dClient.iCnt + 1 ;
				_dClient.iReqId := _dClient.iReqId +1;
				_dClient.TimeOutLeft := _dClient.TimeOut;

				IF _dCltIf.iState = 1 THEN // falls über state dann "schnellwiederholung" aktivieren
					_dClient.iTimeOutCnt := 0; // scharf machen für den nächsten versuch
				END_IF;
				_dCltIf.iState := 2;

				Kanlink.ServerData.HeaderV1Send.Command := _dClient.Cmd;
				Kanlink.ServerData.HeaderV1Send.CmdNr := _dClient.CmdOpt AND 16#000F;

				Kanlink.ServerData.HeaderV1Send.dataFormat := 5;
				Kanlink.ServerData.HeaderV1Send.Length := UDINT_TO_UINT( _dClient.ReqLength);
				Kanlink.ServerData.HeaderV1Send.ReqID := _dClient.iReqId;
				Kanlink.ServerData.HeaderV1Send.Tag		:= _dCltIf.tag;

				KLLib_SendData(ADR(Kanlink),_dClient.AdrDataReq,_dClient.ReqLength,ADR(_dClient.sClientAdr));

				_dClient.xReqPending := TRUE;
				_dClient.iCycleWait := 0;

				Kanlink._xSendClient := FALSE;

				RETURN;

			END_IF;

		END_IF;	// sendClient

#ifndef  HLKANLINK_AUTONOM  // wird MIT Framework gearbeitet
	ELSIF IFmnParam.Out.xParamOK AND IFmnEth.Out.xDataValid THEN

		Kanlink.ServerData.MetaInfoResp.KanLink_Hostname := IFmnEth.Out.IP.sHostname;
		Kanlink.ServerData.MetaInfoResp.Machine_type := WSTRING_TO_STRING(IFmnParam.Out.HeaderVersion.utfMachineType);
		Kanlink.ServerData.MetaInfoResp.DataModelTimeStamp := IFmnParam.Out.HeaderVersion.dtTimestamp;
		Kanlink.ServerData.MetaInfoResp.DataModelVersion := IFmnParam.Out.HeaderVersion.wVersion;

		Kanlink.ServerData.PingResp.KanLink_Hostname := IFmnEth.Out.IP.sHostname;

		_xInitOK := TRUE;

	END_IF
#else  // falls OHNE Framework gearbeitet wird
	ELSIF TRUE THEN
		_xInitOK := TRUE;
	END_IF
#endif

END_PROGRAM

PROGRAM _EXIT

	Kanlink.udp.close.enable	:= TRUE;
	Kanlink.udp.close.ident		:= Kanlink.udp.open.ident;
	Kanlink.udp.close;

END_PROGRAM
```
